LIN {X 0,Y 334.381,Z 572.13,A -85,B 0,C 180,E1 -16692.837,E2 -16692.837} C_VEL
LIN {X 0,Y 335.361,Z 549.408,A -85,B 0,C 180,E1 -16693.333,E2 -16693.333} C_VEL
LIN {X 0,Y 327.108,Z 531.714,A -85,B 0,C 180,E1 -16695.238,E2 -16695.238} C_VEL
LIN {X 0,Y 318.416,Z 515.187,A -85,B 0,C 180,E1 -16697.361,E2 -16697.361} C_VEL
LIN {X 0,Y 310.407,Z 501.402,A -85,B 0,C 180,E1 -16699.456,E2 -16699.456} C_VEL
LIN {X 0,Y 303.46,Z 490.565,A -85,B 0,C 180,E1 -16701.401,E2 -16701.401} C_VEL
LIN {X 0,Y 299.452,Z 484.565,A -85,B 0,C 180,E1 -16702.595,E2 -16702.595} C_VEL
LIN {X 0,Y 295.371,Z 478.736,A -85,B 0,C 180,E1 -16703.869,E2 -16703.869} C_VEL
LIN {X 0,Y 292.684,Z 474.795,A -85,B 0,C 180,E1 -16704.773,E2 -16704.773} C_VEL
LIN {X 0,Y 291.881,Z 473.268,A -85,B 0,C 180,E1 -16705.284,E2 -16705.284} C_VEL
LIN {X 0,Y 291.349,Z 471.542,A -85,B 0,C 180,E1 -16706.167,E2 -16706.167} C_VEL
LIN {X 0,Y 291.334,Z 471.401,A -85,B 0,C 180,E1 -16709.563,E2 -16709.563} C_VEL
LIN {X 0,Y 291.431,Z 471.376,A -85,B 0,C 180,E1 -16713.158,E2 -16713.158} C_VEL
LIN {X 0,Y 291.426,Z 471.42,A -85,B 0,C 180,E1 -16716.403,E2 -16716.403} C_VEL
LIN {X 0,Y 291.453,Z 471.349,A -85,B 0,C 180,E1 -16720.27,E2 -16720.27} C_VEL
LIN {X 0,Y 291.535,Z 471.417,A -85,B 0,C 180,E1 -16724.634,E2 -16724.634} C_VEL
LIN {X 0,Y 291.529,Z 471.42,A -85,B 0,C 180,E1 -16728.88,E2 -16728.88} C_VEL
LIN {X 0,Y 291.682,Z 471.379,A -85,B 0,C 180,E1 -16731.687,E2 -16731.687} C_VEL
LIN {X 0,Y 291.622,Z 471.406,A -85,B 0,C 180,E1 -16734.468,E2 -16734.468} C_VEL
LIN {X 0,Y 291.883,Z 471.376,A -85,B 0,C 180,E1 -16738.62,E2 -16738.62} C_VEL
LIN {X 0,Y 291.883,Z 471.351,A -85,B 0,C 180,E1 -16741.379,E2 -16741.379} C_VEL
LIN {X 0,Y 291.735,Z 471.371,A -85,B 0,C 180,E1 -16746.918,E2 -16746.918} C_VEL
LIN {X 0,Y 291.623,Z 471.396,A -85,B 0,C 180,E1 -16749.712,E2 -16749.712} C_VEL
LIN {X 0,Y 291.515,Z 471.42,A -85,B 0,C 180,E1 -16753.95,E2 -16753.95} C_VEL
LIN {X 0,Y 291.479,Z 471.41,A -85,B 0,C 180,E1 -16756.818,E2 -16756.818} C_VEL
LIN {X 0,Y 291.445,Z 471.415,A -85,B 0,C 180,E1 -16759.875,E2 -16759.875} C_VEL
LIN {X 0,Y 291.375,Z 471.402,A -85,B 0,C 180,E1 -16764.207,E2 -16764.207} C_VEL
LIN {X 0,Y 291.41,Z 471.367,A -85,B 0,C 180,E1 -16767.272,E2 -16767.272} C_VEL
LIN {X 0,Y 291.331,Z 471.448,A -85,B 0,C 180,E1 -16770.437,E2 -16770.437} C_VEL
LIN {X 0,Y 291.361,Z 471.384,A -85,B 0,C 180,E1 -16774.308,E2 -16774.308} C_VEL
LIN {X 0,Y 291.431,Z 471.801,A -85,B 0,C 180,E1 -16774.993,E2 -16774.993} C_VEL
LIN {X 0,Y 291.85,Z 473.233,A -85,B 0,C 180,E1 -16775.358,E2 -16775.358} C_VEL
LIN {X 0,Y 293.498,Z 475.642,A -85,B 0,C 180,E1 -16775.92,E2 -16775.92} C_VEL
LIN {X 0,Y 295.287,Z 477.12,A -85,B 0,C 180,E1 -16776.46,E2 -16776.46} C_VEL
LIN {X 0,Y 297.213,Z 480.287,A -85,B 0,C 180,E1 -16777.088,E2 -16777.088} C_VEL
LIN {X 0,Y 299.738,Z 482.814,A -85,B 0,C 180,E1 -16777.829,E2 -16777.829} C_VEL
LIN {X 0,Y 302.494,Z 486.373,A -85,B 0,C 180,E1 -16778.672,E2 -16778.672} C_VEL
LIN {X 0,Y 304.519,Z 488.28,A -85,B 0,C 180,E1 -16779.288,E2 -16779.288} C_VEL
LIN {X 0,Y 307.616,Z 492.007,A -85,B 0,C 180,E1 -16780.283,E2 -16780.283} C_VEL
LIN {X 0,Y 309.885,Z 494.075,A -85,B 0,C 180,E1 -16781.012,E2 -16781.012} C_VEL
LIN {X 0,Y 313.007,Z 497.745,A -85,B 0,C 180,E1 -16782.091,E2 -16782.091} C_VEL
LIN {X 0,Y 316.165,Z 500.564,A -85,B 0,C 180,E1 -16783.182,E2 -16783.182} C_VEL
LIN {X 0,Y 319.669,Z 504.411,A -85,B 0,C 180,E1 -16784.495,E2 -16784.495} C_VEL
LIN {X 0,Y 321.978,Z 506.47,A -85,B 0,C 180,E1 -16785.384,E2 -16785.384} C_VEL
LIN {X 0,Y 325.336,Z 510.246,A -85,B 0,C 180,E1 -16786.766,E2 -16786.766} C_VEL
LIN {X 0,Y 327.744,Z 512.477,A -85,B 0,C 180,E1 -16787.764,E2 -16787.764} C_VEL
LIN {X 0,Y 331.281,Z 516.359,A -85,B 0,C 180,E1 -16789.27,E2 -16789.27} C_VEL
LIN {X 0,Y 333.728,Z 518.535,A -85,B 0,C 180,E1 -16790.304,E2 -16790.304} C_VEL
LIN {X 0,Y 337.04,Z 522.208,A -85,B 0,C 180,E1 -16791.773,E2 -16791.773} C_VEL
LIN {X 0,Y 339.999,Z 524.765,A -85,B 0,C 180,E1 -16793.076,E2 -16793.076} C_VEL
LIN {X 0,Y 343.638,Z 528.709,A -85,B 0,C 180,E1 -16794.782,E2 -16794.782} C_VEL
LIN {X 0,Y 346.549,Z 531.16,A -85,B 0,C 180,E1 -16796.145,E2 -16796.145} C_VEL
LIN {X 0,Y 350.058,Z 534.897,A -85,B 0,C 180,E1 -16797.894,E2 -16797.894} C_VEL
LIN {X 0,Y 353.412,Z 537.55,A -85,B 0,C 180,E1 -16799.575,E2 -16799.575} C_VEL
LIN {X 0,Y 356.669,Z 541.059,A -85,B 0,C 180,E1 -16801.336,E2 -16801.336} C_VEL
LIN {X 0,Y 360.36,Z 544.044,A -85,B 0,C 180,E1 -16803.41,E2 -16803.41} C_VEL
LIN {X 0,Y 363.49,Z 547.556,A -85,B 0,C 180,E1 -16805.33,E2 -16805.33} C_VEL
LIN {X 0,Y 366.856,Z 549.992,A -85,B 0,C 180,E1 -16807.472,E2 -16807.472} C_VEL
LIN {X 0,Y 367.902,Z 550.793,A -85,B 0,C 180,E1 -16808.161,E2 -16808.161} C_VEL
LIN {X 0,Y 370.532,Z 553.885,A -85,B 0,C 180,E1 -16810.125,E2 -16810.125} C_VEL
LIN {X 0,Y 373.757,Z 556.298,A -85,B 0,C 180,E1 -16812.65,E2 -16812.65} C_VEL
LIN {X 0,Y 375.673,Z 557.433,A -85,B 0,C 180,E1 -16814.324,E2 -16814.324} C_VEL
LIN {X 0,Y 377.714,Z 560.107,A -85,B 0,C 180,E1 -16816.455,E2 -16816.455} C_VEL
LIN {X 0,Y 379.831,Z 562.032,A -85,B 0,C 180,E1 -16819.013,E2 -16819.013} C_VEL
LIN {X 0,Y 381.592,Z 562.974,A -85,B 0,C 180,E1 -16821.527,E2 -16821.527} C_VEL
LIN {X 0,Y 383.034,Z 563.727,A -85,B 0,C 180,E1 -16824.382,E2 -16824.382} C_VEL
LIN {X 0,Y 383.818,Z 564.175,A -85,B 0,C 180,E1 -16826.851,E2 -16826.851} C_VEL
LIN {X 0,Y 384.122,Z 564.361,A -85,B 0,C 180,E1 -16828.952,E2 -16828.952} C_VEL
LIN {X 0,Y 384.122,Z 564.364,A -85,B 0,C 180,E1 -16831.048,E2 -16831.048} C_VEL
LIN {X 0,Y 383.818,Z 564.175,A -85,B 0,C 180,E1 -16833.149,E2 -16833.149} C_VEL
LIN {X 0,Y 383.04,Z 563.678,A -85,B 0,C 180,E1 -16835.617,E2 -16835.617} C_VEL
LIN {X 0,Y 381.59,Z 562.994,A -85,B 0,C 180,E1 -16838.473,E2 -16838.473} C_VEL
LIN {X 0,Y 379.842,Z 561.96,A -85,B 0,C 180,E1 -16840.986,E2 -16840.986} C_VEL
LIN {X 0,Y 377.843,Z 560.265,A -85,B 0,C 180,E1 -16843.385,E2 -16843.385} C_VEL
LIN {X 0,Y 375.673,Z 557.437,A -85,B 0,C 180,E1 -16845.675,E2 -16845.675} C_VEL
LIN {X 0,Y 372.39,Z 555.413,A -85,B 0,C 180,E1 -16848.438,E2 -16848.438} C_VEL
LIN {X 0,Y 369.449,Z 552.788,A -85,B 0,C 180,E1 -16850.683,E2 -16850.683} C_VEL
LIN {X 0,Y 367.271,Z 550.225,A -85,B 0,C 180,E1 -16852.258,E2 -16852.258} C_VEL
LIN {X 0,Y 363.795,Z 547.809,A -85,B 0,C 180,E1 -16854.492,E2 -16854.492} C_VEL
LIN {X 0,Y 360.494,Z 544.264,A -85,B 0,C 180,E1 -16856.507,E2 -16856.507} C_VEL
LIN {X 0,Y 359.349,Z 543.135,A -85,B 0,C 180,E1 -16857.187,E2 -16857.187} C_VEL
LIN {X 0,Y 355.514,Z 540.032,A -85,B 0,C 180,E1 -16859.274,E2 -16859.274} C_VEL
LIN {X 0,Y 352.562,Z 536.779,A -85,B 0,C 180,E1 -16860.861,E2 -16860.861} C_VEL
LIN {X 0,Y 348.845,Z 533.753,A -85,B 0,C 180,E1 -16862.72,E2 -16862.72} C_VEL
LIN {X 0,Y 345.524,Z 530.115,A -85,B 0,C 180,E1 -16864.36,E2 -16864.36} C_VEL
LIN {X 0,Y 341.728,Z 526.843,A -85,B 0,C 180,E1 -16866.11,E2 -16866.11} C_VEL
LIN {X 0,Y 339.088,Z 523.809,A -85,B 0,C 180,E1 -16867.343,E2 -16867.343} C_VEL
LIN {X 0,Y 335.34,Z 520.521,A -85,B 0,C 180,E1 -16868.977,E2 -16868.977} C_VEL
LIN {X 0,Y 332.728,Z 517.523,A -85,B 0,C 180,E1 -16870.137,E2 -16870.137} C_VEL
LIN {X 0,Y 328.735,Z 513.73,A -85,B 0,C 180,E1 -16871.818,E2 -16871.818} C_VEL
LIN {X 0,Y 326.576,Z 511.305,A -85,B 0,C 180,E1 -16872.724,E2 -16872.724} C_VEL
LIN {X 0,Y 322.795,Z 507.577,A -85,B 0,C 180,E1 -16874.272,E2 -16874.272} C_VEL
LIN {X 0,Y 320.948,Z 505.42,A -85,B 0,C 180,E1 -16875.019,E2 -16875.019} C_VEL
LIN {X 0,Y 317.286,Z 501.993,A -85,B 0,C 180,E1 -16876.396,E2 -16876.396} C_VEL
LIN {X 0,Y 315.159,Z 499.492,A -85,B 0,C 180,E1 -16877.182,E2 -16877.182} C_VEL
LIN {X 0,Y 311.478,Z 496.114,A -85,B 0,C 180,E1 -16878.445,E2 -16878.445} C_VEL
LIN {X 0,Y 308.974,Z 493.165,A -85,B 0,C 180,E1 -16879.289,E2 -16879.289} C_VEL
LIN {X 0,Y 305.531,Z 489.71,A -85,B 0,C 180,E1 -16880.387,E2 -16880.387} C_VEL
LIN {X 0,Y 303.826,Z 487.508,A -85,B 0,C 180,E1 -16880.926,E2 -16880.926} C_VEL
LIN {X 0,Y 300.975,Z 484.659,A -85,B 0,C 180,E1 -16881.781,E2 -16881.781} C_VEL
LIN {X 0,Y 299.017,Z 481.929,A -85,B 0,C 180,E1 -16882.39,E2 -16882.39} C_VEL
LIN {X 0,Y 296.451,Z 479.267,A -85,B 0,C 180,E1 -16883.149,E2 -16883.149} C_VEL
LIN {X 0,Y 294.937,Z 476.731,A -85,B 0,C 180,E1 -16883.649,E2 -16883.649} C_VEL
LIN {X 0,Y 292.585,Z 474.553,A -85,B 0,C 180,E1 -16884.374,E2 -16884.374} C_VEL
LIN {X 0,Y 291.469,Z 471.949,A -85,B 0,C 180,E1 -16884.936,E2 -16884.936} C_VEL
LIN {X 0,Y 291.379,Z 471.439,A -85,B 0,C 180,E1 -16885.386,E2 -16885.386} C_VEL
LIN {X 0,Y 291.365,Z 471.403,A -85,B 0,C 180,E1 -16887.951,E2 -16887.951} C_VEL
LIN {X 0,Y 291.371,Z 471.396,A -85,B 0,C 180,E1 -16891.158,E2 -16891.158} C_VEL
LIN {X 0,Y 291.404,Z 471.37,A -85,B 0,C 180,E1 -16894.271,E2 -16894.271} C_VEL
LIN {X 0,Y 291.368,Z 471.442,A -85,B 0,C 180,E1 -16897.299,E2 -16897.299} C_VEL
LIN {X 0,Y 291.452,Z 471.414,A -85,B 0,C 180,E1 -16900.27,E2 -16900.27} C_VEL
LIN {X 0,Y 291.534,Z 471.399,A -85,B 0,C 180,E1 -16904.635,E2 -16904.635} C_VEL
LIN {X 0,Y 291.529,Z 471.397,A -85,B 0,C 180,E1 -16908.881,E2 -16908.881} C_VEL
LIN {X 0,Y 291.7,Z 471.394,A -85,B 0,C 180,E1 -16911.689,E2 -16911.689} C_VEL
LIN {X 0,Y 291.623,Z 471.389,A -85,B 0,C 180,E1 -16914.469,E2 -16914.469} C_VEL
LIN {X 0,Y 291.883,Z 471.353,A -85,B 0,C 180,E1 -16918.621,E2 -16918.621} C_VEL
LIN {X 0,Y 291.883,Z 471.377,A -85,B 0,C 180,E1 -16921.38,E2 -16921.38} C_VEL
LIN {X 0,Y 291.73,Z 471.386,A -85,B 0,C 180,E1 -16926.919,E2 -16926.919} C_VEL
LIN {X 0,Y 291.569,Z 471.399,A -85,B 0,C 180,E1 -16929.714,E2 -16929.714} C_VEL
LIN {X 0,Y 291.511,Z 471.402,A -85,B 0,C 180,E1 -16933.879,E2 -16933.879} C_VEL
LIN {X 0,Y 290.876,Z 471.497,A -85,B 0,C 180,E1 -16935.032,E2 -16935.032} C_VEL
LIN {X 0,Y 287.965,Z 471.838,A -85,B 0,C 180,E1 -16936.906,E2 -16936.906} C_VEL
LIN {X 0,Y 285.485,Z 472.113,A -85,B 0,C 180,E1 -16938.428,E2 -16938.428} C_VEL
LIN {X 0,Y 284.446,Z 472.222,A -85,B 0,C 180,E1 -16939.61,E2 -16939.61} C_VEL
LIN {X 0,Y 284.378,Z 472.229,A -85,B 0,C 180,E1 -16940.01,E2 -16940.01} C_VEL
LIN {X 0,Y 284.37,Z 472.306,A -85,B 0,C 180,E1 -16943.878,E2 -16943.878} C_VEL
LIN {X 0,Y 284.388,Z 472.248,A -85,B 0,C 180,E1 -16947.172,E2 -16947.172} C_VEL
LIN {X 0,Y 284.306,Z 472.298,A -85,B 0,C 180,E1 -16951.273,E2 -16951.273} C_VEL
LIN {X 0,Y 284.379,Z 472.631,A -85,B 0,C 180,E1 -16952.385,E2 -16952.385} C_VEL
LIN {X 0,Y 284.771,Z 474.121,A -85,B 0,C 180,E1 -16952.885,E2 -16952.885} C_VEL
LIN {X 0,Y 286.497,Z 476.648,A -85,B 0,C 180,E1 -16953.552,E2 -16953.552} C_VEL
LIN {X 0,Y 289.794,Z 480.785,A -85,B 0,C 180,E1 -16954.692,E2 -16954.692} C_VEL
LIN {X 0,Y 294.042,Z 486.894,A -85,B 0,C 180,E1 -16956.109,E2 -16956.109} C_VEL
LIN {X 0,Y 297.851,Z 492.54,A -85,B 0,C 180,E1 -16957.314,E2 -16957.314} C_VEL
LIN {X 0,Y 304.433,Z 502.659,A -85,B 0,C 180,E1 -16959.268,E2 -16959.268} C_VEL
LIN {X 0,Y 312.901,Z 517.15,A -85,B 0,C 180,E1 -16961.605,E2 -16961.605} C_VEL
LIN {X 0,Y 320.685,Z 531.778,A -85,B 0,C 180,E1 -16963.603,E2 -16963.603} C_VEL
LIN {X 0,Y 328.783,Z 548.886,A -85,B 0,C 180,E1 -16965.568,E2 -16965.568} C_VEL
LIN {X 0,Y 330.101,Z 551.932,A -85,B 0,C 180,E1 -16965.881,E2 -16965.881} C_VEL
LIN {X 0,Y 324.783,Z 665.436,A -85,B 0,C 180,E1 -16968.34,E2 -16968.34} C_VEL
LIN {X 0,Y 323.346,Z 691.603,A -85,B 0,C 180,E1 -16968.944,E2 -16968.944} C_VEL
LIN {X 0,Y 321.431,Z 710.108,A -85,B 0,C 180,E1 -16969.578,E2 -16969.578} C_VEL
LIN {X 0,Y 319.225,Z 725.277,A -85,B 0,C 180,E1 -16970.324,E2 -16970.324} C_VEL
LIN {X 0,Y 317.056,Z 738.026,A -85,B 0,C 180,E1 -16971.123,E2 -16971.123} C_VEL
LIN {X 0,Y 314.499,Z 750.717,A -85,B 0,C 180,E1 -16972.083,E2 -16972.083} C_VEL
LIN {X 0,Y 311.899,Z 762.357,A -85,B 0,C 180,E1 -16973.135,E2 -16973.135} C_VEL
LIN {X 0,Y 308.638,Z 775.182,A -85,B 0,C 180,E1 -16974.504,E2 -16974.504} C_VEL
LIN {X 0,Y 305.867,Z 785.571,A -85,B 0,C 180,E1 -16975.81,E2 -16975.81} C_VEL
LIN {X 0,Y 302.784,Z 796.148,A -85,B 0,C 180,E1 -16977.34,E2 -16977.34} C_VEL
LIN {X 0,Y 299.815,Z 805.837,A -85,B 0,C 180,E1 -16978.956,E2 -16978.956} C_VEL
LIN {X 0,Y 297.116,Z 814.636,A -85,B 0,C 180,E1 -16980.645,E2 -16980.645} C_VEL
LIN {X 0,Y 293.939,Z 825.009,A -85,B 0,C 180,E1 -16982.982,E2 -16982.982} C_VEL
LIN {X 0,Y 291.351,Z 832.898,A -85,B 0,C 180,E1 -16985.031,E2 -16985.031} C_VEL
LIN {X 0,Y 289.186,Z 839.864,A -85,B 0,C 180,E1 -16987.118,E2 -16987.118} C_VEL
LIN {X 0,Y 287.414,Z 846.008,A -85,B 0,C 180,E1 -16989.234,E2 -16989.234} C_VEL
LIN {X 0,Y 285.468,Z 852.957,A -85,B 0,C 180,E1 -16992.077,E2 -16992.077} C_VEL
LIN {X 0,Y 284.218,Z 858.207,A -85,B 0,C 180,E1 -16994.659,E2 -16994.659} C_VEL
LIN {X 0,Y 283.341,Z 862.335,A -85,B 0,C 180,E1 -16997.101,E2 -16997.101} C_VEL
LIN {X 0,Y 282.63,Z 866.188,A -85,B 0,C 180,E1 -16999.976,E2 -16999.976} C_VEL
LIN {X 0,Y 282.387,Z 869.045,A -85,B 0,C 180,E1 -17002.852,E2 -17002.852} C_VEL
LIN {X 0,Y 282.334,Z 870.439,A -85,B 0,C 180,E1 -17004.682,E2 -17004.682} C_VEL
LIN {X 0,Y 282.329,Z 871.61,A -85,B 0,C 180,E1 -17007.146,E2 -17007.146} C_VEL
LIN {X 0,Y 282.315,Z 872.083,A -85,B 0,C 180,E1 -17010,E2 -17010} C_VEL
LIN {X 0,Y 282.329,Z 871.61,A -85,B 0,C 180,E1 -17012.854,E2 -17012.854} C_VEL
LIN {X 0,Y 282.336,Z 870.182,A -85,B 0,C 180,E1 -17015.714,E2 -17015.714} C_VEL
LIN {X 0,Y 282.482,Z 867.793,A -85,B 0,C 180,E1 -17018.585,E2 -17018.585} C_VEL
LIN {X 0,Y 283.113,Z 863.375,A -85,B 0,C 180,E1 -17022.181,E2 -17022.181} C_VEL
LIN {X 0,Y 283.809,Z 860.006,A -85,B 0,C 180,E1 -17024.337,E2 -17024.337} C_VEL
LIN {X 0,Y 285.075,Z 854.503,A -85,B 0,C 180,E1 -17027.207,E2 -17027.207} C_VEL
LIN {X 0,Y 286.406,Z 849.643,A -85,B 0,C 180,E1 -17029.345,E2 -17029.345} C_VEL
LIN {X 0,Y 288.683,Z 841.563,A -85,B 0,C 180,E1 -17032.315,E2 -17032.315} C_VEL
LIN {X 0,Y 290.552,Z 835.315,A -85,B 0,C 180,E1 -17034.28,E2 -17034.28} C_VEL
LIN {X 0,Y 293.007,Z 827.765,A -85,B 0,C 180,E1 -17036.342,E2 -17036.342} C_VEL
LIN {X 0,Y 295.883,Z 818.635,A -85,B 0,C 180,E1 -17038.497,E2 -17038.497} C_VEL
LIN {X 0,Y 298.73,Z 809.388,A -85,B 0,C 180,E1 -17040.385,E2 -17040.385} C_VEL
LIN {X 0,Y 301.849,Z 799.167,A -85,B 0,C 180,E1 -17042.181,E2 -17042.181} C_VEL
LIN {X 0,Y 304.936,Z 788.746,A -85,B 0,C 180,E1 -17043.755,E2 -17043.755} C_VEL
LIN {X 0,Y 307.943,Z 777.792,A -85,B 0,C 180,E1 -17045.187,E2 -17045.187} C_VEL
LIN {X 0,Y 310.748,Z 766.854,A -85,B 0,C 180,E1 -17046.418,E2 -17046.418} C_VEL
LIN {X 0,Y 313.345,Z 755.941,A -85,B 0,C 180,E1 -17047.472,E2 -17047.472} C_VEL
LIN {X 0,Y 316.032,Z 743.211,A -85,B 0,C 180,E1 -17048.51,E2 -17048.51} C_VEL
LIN {X 0,Y 318.448,Z 730.004,A -85,B 0,C 180,E1 -17049.399,E2 -17049.399} C_VEL
LIN {X 0,Y 320.485,Z 717.004,A -85,B 0,C 180,E1 -17050.103,E2 -17050.103} C_VEL
LIN {X 0,Y 322.187,Z 703.636,A -85,B 0,C 180,E1 -17050.667,E2 -17050.667} C_VEL
LIN {X 0,Y 323.432,Z 690.183,A -85,B 0,C 180,E1 -17051.094,E2 -17051.094} C_VEL
LIN {X 0,Y 325.351,Z 652.898,A -85,B 0,C 180,E1 -17051.934,E2 -17051.934} C_VEL
LIN {X 0,Y 330.17,Z 552.059,A -85,B 0,C 180,E1 -17054.104,E2 -17054.104} C_VEL
LIN {X 0,Y 322.6,Z 535.681,A -85,B 0,C 180,E1 -17055.922,E2 -17055.922} C_VEL
LIN {X 0,Y 314.412,Z 519.91,A -85,B 0,C 180,E1 -17057.996,E2 -17057.996} C_VEL
LIN {X 0,Y 306.931,Z 506.798,A -85,B 0,C 180,E1 -17060.022,E2 -17060.022} C_VEL
LIN {X 0,Y 300.04,Z 495.907,A -85,B 0,C 180,E1 -17062.018,E2 -17062.018} C_VEL
LIN {X 0,Y 296.102,Z 489.901,A -85,B 0,C 180,E1 -17063.234,E2 -17063.234} C_VEL
LIN {X 0,Y 292.28,Z 484.386,A -85,B 0,C 180,E1 -17064.467,E2 -17064.467} C_VEL
LIN {X 0,Y 288.574,Z 479.142,A -85,B 0,C 180,E1 -17065.728,E2 -17065.728} C_VEL
LIN {X 0,Y 284.924,Z 474.496,A -85,B 0,C 180,E1 -17067.041,E2 -17067.041} C_VEL
LIN {X 0,Y 284.431,Z 472.918,A -85,B 0,C 180,E1 -17067.477,E2 -17067.477} C_VEL
LIN {X 0,Y 284.376,Z 472.392,A -85,B 0,C 180,E1 -17067.903,E2 -17067.903} C_VEL
LIN {X 0,Y 284.321,Z 472.249,A -85,B 0,C 180,E1 -17071.988,E2 -17071.988} C_VEL
LIN {X 0,Y 284.347,Z 472.31,A -85,B 0,C 180,E1 -17075.154,E2 -17075.154} C_VEL
LIN {X 0,Y 284.31,Z 472.252,A -85,B 0,C 180,E1 -17078.235,E2 -17078.235} C_VEL
LIN {X 0,Y 284.392,Z 472.236,A -85,B 0,C 180,E1 -17081.261,E2 -17081.261} C_VEL
LIN {X 0,Y 284.473,Z 472.298,A -85,B 0,C 180,E1 -17084.469,E2 -17084.469} C_VEL
LIN {X 0,Y 284.481,Z 472.294,A -85,B 0,C 180,E1 -17088.601,E2 -17088.601} C_VEL
LIN {X 0,Y 284.633,Z 472.256,A -85,B 0,C 180,E1 -17091.48,E2 -17091.48} C_VEL
LIN {X 0,Y 284.593,Z 472.283,A -85,B 0,C 180,E1 -17094.331,E2 -17094.331} C_VEL
LIN {X 0,Y 284.849,Z 472.251,A -85,B 0,C 180,E1 -17098.586,E2 -17098.586} C_VEL
LIN {X 0,Y 284.849,Z 472.226,A -85,B 0,C 180,E1 -17101.413,E2 -17101.413} C_VEL
LIN {X 0,Y 284.688,Z 472.249,A -85,B 0,C 180,E1 -17107.09,E2 -17107.09} C_VEL
LIN {X 0,Y 284.56,Z 472.271,A -85,B 0,C 180,E1 -17109.955,E2 -17109.955} C_VEL
LIN {X 0,Y 284.472,Z 472.29,A -85,B 0,C 180,E1 -17114.303,E2 -17114.303} C_VEL
LIN {X 0,Y 284.416,Z 472.295,A -85,B 0,C 180,E1 -17117.248,E2 -17117.248} C_VEL
LIN {X 0,Y 284.371,Z 472.294,A -85,B 0,C 180,E1 -17120.242,E2 -17120.242} C_VEL
LIN {X 0,Y 284.329,Z 472.262,A -85,B 0,C 180,E1 -17124.847,E2 -17124.847} C_VEL
LIN {X 0,Y 284.319,Z 472.256,A -85,B 0,C 180,E1 -17128.011,E2 -17128.011} C_VEL
LIN {X 0,Y 284.345,Z 472.276,A -85,B 0,C 180,E1 -17132.041,E2 -17132.041} C_VEL
LIN {X 0,Y 284.336,Z 472.559,A -85,B 0,C 180,E1 -17132.821,E2 -17132.821} C_VEL
LIN {X 0,Y 284.661,Z 473.798,A -85,B 0,C 180,E1 -17133.268,E2 -17133.268} C_VEL
LIN {X 0,Y 286.187,Z 476.255,A -85,B 0,C 180,E1 -17133.858,E2 -17133.858} C_VEL
LIN {X 0,Y 288.455,Z 478.173,A -85,B 0,C 180,E1 -17134.612,E2 -17134.612} C_VEL
LIN {X 0,Y 290.288,Z 481.161,A -85,B 0,C 180,E1 -17135.263,E2 -17135.263} C_VEL
LIN {X 0,Y 292.472,Z 483.386,A -85,B 0,C 180,E1 -17135.96,E2 -17135.96} C_VEL
LIN {X 0,Y 295.096,Z 487.032,A -85,B 0,C 180,E1 -17136.808,E2 -17136.808} C_VEL
LIN {X 0,Y 296.858,Z 488.838,A -85,B 0,C 180,E1 -17137.334,E2 -17137.334} C_VEL
LIN {X 0,Y 299.815,Z 492.532,A -85,B 0,C 180,E1 -17138.232,E2 -17138.232} C_VEL
LIN {X 0,Y 301.873,Z 494.497,A -85,B 0,C 180,E1 -17138.836,E2 -17138.836} C_VEL
LIN {X 0,Y 305.432,Z 498.533,A -85,B 0,C 180,E1 -17139.95,E2 -17139.95} C_VEL
LIN {X 0,Y 307.628,Z 500.638,A -85,B 0,C 180,E1 -17140.646,E2 -17140.646} C_VEL
LIN {X 0,Y 311.443,Z 504.735,A -85,B 0,C 180,E1 -17141.927,E2 -17141.927} C_VEL
LIN {X 0,Y 314.013,Z 507.046,A -85,B 0,C 180,E1 -17142.798,E2 -17142.798} C_VEL
LIN {X 0,Y 317.607,Z 510.88,A -85,B 0,C 180,E1 -17144.118,E2 -17144.118} C_VEL
LIN {X 0,Y 319.983,Z 512.995,A -85,B 0,C 180,E1 -17145.011,E2 -17145.011} C_VEL
LIN {X 0,Y 323.545,Z 516.875,A -85,B 0,C 180,E1 -17146.453,E2 -17146.453} C_VEL
LIN {X 0,Y 325.996,Z 519.227,A -85,B 0,C 180,E1 -17147.459,E2 -17147.459} C_VEL
LIN {X 0,Y 329.92,Z 523.309,A -85,B 0,C 180,E1 -17149.112,E2 -17149.112} C_VEL
LIN {X 0,Y 331.953,Z 525.148,A -85,B 0,C 180,E1 -17149.958,E2 -17149.958} C_VEL
LIN {X 0,Y 335.766,Z 529.203,A -85,B 0,C 180,E1 -17151.636,E2 -17151.636} C_VEL
LIN {X 0,Y 338.425,Z 531.541,A -85,B 0,C 180,E1 -17152.804,E2 -17152.804} C_VEL
LIN {X 0,Y 342.225,Z 535.55,A -85,B 0,C 180,E1 -17154.564,E2 -17154.564} C_VEL
LIN {X 0,Y 345.179,Z 538.054,A -85,B 0,C 180,E1 -17155.94,E2 -17155.94} C_VEL
LIN {X 0,Y 348.729,Z 541.782,A -85,B 0,C 180,E1 -17157.702,E2 -17157.702} C_VEL
LIN {X 0,Y 351.946,Z 544.324,A -85,B 0,C 180,E1 -17159.307,E2 -17159.307} C_VEL
LIN {X 0,Y 355.165,Z 547.781,A -85,B 0,C 180,E1 -17161.037,E2 -17161.037} C_VEL
LIN {X 0,Y 359.171,Z 551.025,A -85,B 0,C 180,E1 -17163.254,E2 -17163.254} C_VEL
LIN {X 0,Y 362.444,Z 554.622,A -85,B 0,C 180,E1 -17165.254,E2 -17165.254} C_VEL
LIN {X 0,Y 366.069,Z 557.131,A -85,B 0,C 180,E1 -17167.544,E2 -17167.544} C_VEL
LIN {X 0,Y 369.45,Z 560.835,A -85,B 0,C 180,E1 -17169.977,E2 -17169.977} C_VEL
LIN {X 0,Y 372.6,Z 563.185,A -85,B 0,C 180,E1 -17172.435,E2 -17172.435} C_VEL
LIN {X 0,Y 374.66,Z 564.449,A -85,B 0,C 180,E1 -17174.201,E2 -17174.201} C_VEL
LIN {X 0,Y 376.8,Z 567.179,A -85,B 0,C 180,E1 -17176.421,E2 -17176.421} C_VEL
LIN {X 0,Y 378.934,Z 569.079,A -85,B 0,C 180,E1 -17178.987,E2 -17178.987} C_VEL
LIN {X 0,Y 380.71,Z 570.019,A -85,B 0,C 180,E1 -17181.508,E2 -17181.508} C_VEL
LIN {X 0,Y 382.002,Z 570.622,A -85,B 0,C 180,E1 -17184.011,E2 -17184.011} C_VEL
LIN {X 0,Y 382.654,Z 571.132,A -85,B 0,C 180,E1 -17185.787,E2 -17185.787} C_VEL
LIN {X 0,Y 383.151,Z 571.293,A -85,B 0,C 180,E1 -17187.898,E2 -17187.898} C_VEL
LIN {X 0,Y 383.34,Z 571.349,A -85,B 0,C 180,E1 -17190,E2 -17190} C_VEL
LIN {X 0,Y 383.151,Z 571.294,A -85,B 0,C 180,E1 -17192.102,E2 -17192.102} C_VEL
LIN {X 0,Y 382.496,Z 571.028,A -85,B 0,C 180,E1 -17194.694,E2 -17194.694} C_VEL
LIN {X 0,Y 381.321,Z 570.322,A -85,B 0,C 180,E1 -17197.412,E2 -17197.412} C_VEL
LIN {X 0,Y 379.645,Z 569.506,A -85,B 0,C 180,E1 -17200.07,E2 -17200.07} C_VEL
LIN {X 0,Y 377.507,Z 567.926,A -85,B 0,C 180,E1 -17202.74,E2 -17202.74} C_VEL
LIN {X 0,Y 375.425,Z 565.498,A -85,B 0,C 180,E1 -17205.035,E2 -17205.035} C_VEL
LIN {X 0,Y 374.396,Z 564.104,A -85,B 0,C 180,E1 -17206.05,E2 -17206.05} C_VEL
LIN {X 0,Y 371.444,Z 562.454,A -85,B 0,C 180,E1 -17208.487,E2 -17208.487} C_VEL
LIN {X 0,Y 368.378,Z 559.8,A -85,B 0,C 180,E1 -17210.8,E2 -17210.8} C_VEL
LIN {X 0,Y 366.07,Z 557.136,A -85,B 0,C 180,E1 -17212.457,E2 -17212.457} C_VEL
LIN {X 0,Y 362.446,Z 554.612,A -85,B 0,C 180,E1 -17214.747,E2 -17214.747} C_VEL
LIN {X 0,Y 359.063,Z 550.952,A -85,B 0,C 180,E1 -17216.81,E2 -17216.81} C_VEL
LIN {X 0,Y 357.753,Z 549.797,A -85,B 0,C 180,E1 -17217.555,E2 -17217.555} C_VEL
LIN {X 0,Y 353.873,Z 546.58,A -85,B 0,C 180,E1 -17219.658,E2 -17219.658} C_VEL
LIN {X 0,Y 351.189,Z 543.603,A -85,B 0,C 180,E1 -17221.088,E2 -17221.088} C_VEL
LIN {X 0,Y 347.28,Z 540.406,A -85,B 0,C 180,E1 -17223.021,E2 -17223.021} C_VEL
LIN {X 0,Y 343.964,Z 536.89,A -85,B 0,C 180,E1 -17224.633,E2 -17224.633} C_VEL
LIN {X 0,Y 339.964,Z 533.38,A -85,B 0,C 180,E1 -17226.47,E2 -17226.47} C_VEL
LIN {X 0,Y 337.366,Z 530.449,A -85,B 0,C 180,E1 -17227.664,E2 -17227.664} C_VEL
LIN {X 0,Y 333.548,Z 527.09,A -85,B 0,C 180,E1 -17229.322,E2 -17229.322} C_VEL
LIN {X 0,Y 331.011,Z 524.2,A -85,B 0,C 180,E1 -17230.438,E2 -17230.438} C_VEL
LIN {X 0,Y 327.099,Z 520.525,A -85,B 0,C 180,E1 -17232.073,E2 -17232.073} C_VEL
LIN {X 0,Y 324.66,Z 517.809,A -85,B 0,C 180,E1 -17233.105,E2 -17233.105} C_VEL
LIN {X 0,Y 320.712,Z 513.934,A -85,B 0,C 180,E1 -17234.695,E2 -17234.695} C_VEL
LIN {X 0,Y 318.781,Z 511.796,A -85,B 0,C 180,E1 -17235.455,E2 -17235.455} C_VEL
LIN {X 0,Y 314.829,Z 508.059,A -85,B 0,C 180,E1 -17236.899,E2 -17236.899} C_VEL
LIN {X 0,Y 312.794,Z 505.825,A -85,B 0,C 180,E1 -17237.62,E2 -17237.62} C_VEL
LIN {X 0,Y 308.869,Z 502.157,A -85,B 0,C 180,E1 -17238.936,E2 -17238.936} C_VEL
LIN {X 0,Y 306.435,Z 499.394,A -85,B 0,C 180,E1 -17239.737,E2 -17239.737} C_VEL
LIN {X 0,Y 302.72,Z 495.657,A -85,B 0,C 180,E1 -17240.891,E2 -17240.891} C_VEL
LIN {X 0,Y 300.986,Z 493.546,A -85,B 0,C 180,E1 -17241.432,E2 -17241.432} C_VEL
LIN {X 0,Y 297.587,Z 489.944,A -85,B 0,C 180,E1 -17242.438,E2 -17242.438} C_VEL
LIN {X 0,Y 295.872,Z 487.752,A -85,B 0,C 180,E1 -17242.962,E2 -17242.962} C_VEL
LIN {X 0,Y 293.13,Z 484.531,A -85,B 0,C 180,E1 -17243.815,E2 -17243.815} C_VEL
LIN {X 0,Y 292.021,Z 482.764,A -85,B 0,C 180,E1 -17244.189,E2 -17244.189} C_VEL
LIN {X 0,Y 289.471,Z 480.074,A -85,B 0,C 180,E1 -17245.015,E2 -17245.015} C_VEL
LIN {X 0,Y 288.027,Z 477.677,A -85,B 0,C 180,E1 -17245.534,E2 -17245.534} C_VEL
LIN {X 0,Y 285.644,Z 475.624,A -85,B 0,C 180,E1 -17246.334,E2 -17246.334} C_VEL
LIN {X 0,Y 284.393,Z 472.94,A -85,B 0,C 180,E1 -17246.961,E2 -17246.961} C_VEL
LIN {X 0,Y 284.31,Z 472.32,A -85,B 0,C 180,E1 -17247.446,E2 -17247.446} C_VEL
LIN {X 0,Y 284.352,Z 472.29,A -85,B 0,C 180,E1 -17250.376,E2 -17250.376} C_VEL
LIN {X 0,Y 284.367,Z 472.24,A -85,B 0,C 180,E1 -17253.586,E2 -17253.586} C_VEL
LIN {X 0,Y 284.327,Z 472.306,A -85,B 0,C 180,E1 -17256.704,E2 -17256.704} C_VEL
LIN {X 0,Y 284.393,Z 472.305,A -85,B 0,C 180,E1 -17261.261,E2 -17261.261} C_VEL
LIN {X 0,Y 284.472,Z 472.278,A -85,B 0,C 180,E1 -17264.47,E2 -17264.47} C_VEL
LIN {X 0,Y 284.481,Z 472.274,A -85,B 0,C 180,E1 -17268.602,E2 -17268.602} C_VEL
LIN {X 0,Y 284.65,Z 472.274,A -85,B 0,C 180,E1 -17271.481,E2 -17271.481} C_VEL
LIN {X 0,Y 284.593,Z 472.263,A -85,B 0,C 180,E1 -17274.331,E2 -17274.331} C_VEL
LIN {X 0,Y 284.849,Z 472.229,A -85,B 0,C 180,E1 -17278.587,E2 -17278.587} C_VEL
LIN {X 0,Y 284.849,Z 472.253,A -85,B 0,C 180,E1 -17281.414,E2 -17281.414} C_VEL
LIN {X 0,Y 284.681,Z 472.261,A -85,B 0,C 180,E1 -17287.091,E2 -17287.091} C_VEL
LIN {X 0,Y 284.513,Z 472.28,A -85,B 0,C 180,E1 -17289.957,E2 -17289.957} C_VEL
LIN {X 0,Y 284.472,Z 472.282,A -85,B 0,C 180,E1 -17294.303,E2 -17294.303} C_VEL
LIN {X 0,Y 284.417,Z 472.267,A -85,B 0,C 180,E1 -17297.249,E2 -17297.249} C_VEL
LIN {X 0,Y 284.378,Z 472.229,A -85,B 0,C 180,E1 -17300.01,E2 -17300.01} C_VEL
LIN {X 0,Y 283.743,Z 472.319,A -85,B 0,C 180,E1 -17301.193,E2 -17301.193} C_VEL
LIN {X 0,Y 280.867,Z 472.714,A -85,B 0,C 180,E1 -17303.119,E2 -17303.119} C_VEL
LIN {X 0,Y 278.414,Z 473.052,A -85,B 0,C 180,E1 -17304.683,E2 -17304.683} C_VEL
LIN {X 0,Y 277.376,Z 473.146,A -85,B 0,C 180,E1 -17305.896,E2 -17305.896} C_VEL
LIN {X 0,Y 277.302,Z 473.143,A -85,B 0,C 180,E1 -17306.307,E2 -17306.307} C_VEL
LIN {X 0,Y 277.308,Z 473.311,A -85,B 0,C 180,E1 -17310.036,E2 -17310.036} C_VEL
LIN {X 0,Y 277.499,Z 474.28,A -85,B 0,C 180,E1 -17310.495,E2 -17310.495} C_VEL
LIN {X 0,Y 279.005,Z 477.022,A -85,B 0,C 180,E1 -17311.195,E2 -17311.195} C_VEL
LIN {X 0,Y 281.492,Z 479.087,A -85,B 0,C 180,E1 -17312.111,E2 -17312.111} C_VEL
LIN {X 0,Y 283.387,Z 482.182,A -85,B 0,C 180,E1 -17312.853,E2 -17312.853} C_VEL
LIN {X 0,Y 286.842,Z 486.535,A -85,B 0,C 180,E1 -17314.088,E2 -17314.088} C_VEL
LIN {X 0,Y 291.131,Z 492.765,A -85,B 0,C 180,E1 -17315.565,E2 -17315.565} C_VEL
LIN {X 0,Y 294.993,Z 498.661,A -85,B 0,C 180,E1 -17316.828,E2 -17316.828} C_VEL
LIN {X 0,Y 301.438,Z 508.787,A -85,B 0,C 180,E1 -17318.799,E2 -17318.799} C_VEL
LIN {X 0,Y 309.143,Z 522.237,A -85,B 0,C 180,E1 -17320.997,E2 -17320.997} C_VEL
LIN {X 0,Y 316.753,Z 536.757,A -85,B 0,C 180,E1 -17323.018,E2 -17323.018} C_VEL
LIN {X 0,Y 324.404,Z 553.16,A -85,B 0,C 180,E1 -17324.941,E2 -17324.941} C_VEL
LIN {X 0,Y 324.895,Z 554.301,A -85,B 0,C 180,E1 -17325.062,E2 -17325.062} C_VEL
LIN {X 0,Y 319.63,Z 663.437,A -85,B 0,C 180,E1 -17327.459,E2 -17327.459} C_VEL
LIN {X 0,Y 318.024,Z 691.393,A -85,B 0,C 180,E1 -17328.103,E2 -17328.103} C_VEL
LIN {X 0,Y 316.048,Z 709.898,A -85,B 0,C 180,E1 -17328.742,E2 -17328.742} C_VEL
LIN {X 0,Y 313.781,Z 725.067,A -85,B 0,C 180,E1 -17329.494,E2 -17329.494} C_VEL
LIN {X 0,Y 311.442,Z 738.342,A -85,B 0,C 180,E1 -17330.339,E2 -17330.339} C_VEL
LIN {X 0,Y 308.898,Z 750.506,A -85,B 0,C 180,E1 -17331.269,E2 -17331.269} C_VEL
LIN {X 0,Y 306.184,Z 762.145,A -85,B 0,C 180,E1 -17332.329,E2 -17332.329} C_VEL
LIN {X 0,Y 302.85,Z 774.971,A -85,B 0,C 180,E1 -17333.719,E2 -17333.719} C_VEL
LIN {X 0,Y 299.674,Z 786.281,A -85,B 0,C 180,E1 -17335.167,E2 -17335.167} C_VEL
LIN {X 0,Y 296.44,Z 796.942,A -85,B 0,C 180,E1 -17336.754,E2 -17336.754} C_VEL
LIN {X 0,Y 293.081,Z 807.399,A -85,B 0,C 180,E1 -17338.564,E2 -17338.564} C_VEL
LIN {X 0,Y 290.373,Z 815.833,A -85,B 0,C 180,E1 -17340.254,E2 -17340.254} C_VEL
LIN {X 0,Y 287.511,Z 824.795,A -85,B 0,C 180,E1 -17342.327,E2 -17342.327} C_VEL
LIN {X 0,Y 284.798,Z 832.684,A -85,B 0,C 180,E1 -17344.416,E2 -17344.416} C_VEL
LIN {X 0,Y 282.544,Z 839.65,A -85,B 0,C 180,E1 -17346.548,E2 -17346.548} C_VEL
LIN {X 0,Y 280.673,Z 845.794,A -85,B 0,C 180,E1 -17348.711,E2 -17348.711} C_VEL
LIN {X 0,Y 278.624,Z 852.744,A -85,B 0,C 180,E1 -17351.622,E2 -17351.622} C_VEL
LIN {X 0,Y 277.191,Z 858.342,A -85,B 0,C 180,E1 -17354.465,E2 -17354.465} C_VEL
LIN {X 0,Y 276.322,Z 862.122,A -85,B 0,C 180,E1 -17356.768,E2 -17356.768} C_VEL
LIN {X 0,Y 275.572,Z 865.976,A -85,B 0,C 180,E1 -17359.716,E2 -17359.716} C_VEL
LIN {X 0,Y 275.294,Z 868.833,A -85,B 0,C 180,E1 -17362.667,E2 -17362.667} C_VEL
LIN {X 0,Y 275.238,Z 870.332,A -85,B 0,C 180,E1 -17364.768,E2 -17364.768} C_VEL
LIN {X 0,Y 275.239,Z 871.4,A -85,B 0,C 180,E1 -17367.073,E2 -17367.073} C_VEL
LIN {X 0,Y 275.238,Z 871.874,A -85,B 0,C 180,E1 -17370,E2 -17370} C_VEL
LIN {X 0,Y 275.239,Z 871.4,A -85,B 0,C 180,E1 -17372.927,E2 -17372.927} C_VEL
LIN {X 0,Y 275.235,Z 869.971,A -85,B 0,C 180,E1 -17375.862,E2 -17375.862} C_VEL
LIN {X 0,Y 275.402,Z 867.581,A -85,B 0,C 180,E1 -17378.807,E2 -17378.807} C_VEL
LIN {X 0,Y 276.09,Z 863.163,A -85,B 0,C 180,E1 -17382.496,E2 -17382.496} C_VEL
LIN {X 0,Y 276.836,Z 859.794,A -85,B 0,C 180,E1 -17384.706,E2 -17384.706} C_VEL
LIN {X 0,Y 278.181,Z 854.289,A -85,B 0,C 180,E1 -17387.648,E2 -17387.648} C_VEL
LIN {X 0,Y 279.615,Z 849.43,A -85,B 0,C 180,E1 -17389.835,E2 -17389.835} C_VEL
LIN {X 0,Y 282.075,Z 841.135,A -85,B 0,C 180,E1 -17392.946,E2 -17392.946} C_VEL
LIN {X 0,Y 284.403,Z 833.893,A -85,B 0,C 180,E1 -17395.231,E2 -17395.231} C_VEL
LIN {X 0,Y 286.588,Z 827.553,A -85,B 0,C 180,E1 -17396.979,E2 -17396.979} C_VEL
LIN {X 0,Y 289.387,Z 818.966,A -85,B 0,C 180,E1 -17399.059,E2 -17399.059} C_VEL
LIN {X 0,Y 292.529,Z 809.175,A -85,B 0,C 180,E1 -17401.099,E2 -17401.099} C_VEL
LIN {X 0,Y 295.799,Z 798.955,A -85,B 0,C 180,E1 -17402.921,E2 -17402.921} C_VEL
LIN {X 0,Y 299.05,Z 788.344,A -85,B 0,C 180,E1 -17404.546,E2 -17404.546} C_VEL
LIN {X 0,Y 302.113,Z 777.58,A -85,B 0,C 180,E1 -17405.971,E2 -17405.971} C_VEL
LIN {X 0,Y 305.016,Z 766.643,A -85,B 0,C 180,E1 -17407.216,E2 -17407.216} C_VEL
LIN {X 0,Y 308.089,Z 753.988,A -85,B 0,C 180,E1 -17408.433,E2 -17408.433} C_VEL
LIN {X 0,Y 310.723,Z 741.818,A -85,B 0,C 180,E1 -17409.414,E2 -17409.414} C_VEL
LIN {X 0,Y 313.01,Z 729.634,A -85,B 0,C 180,E1 -17410.235,E2 -17410.235} C_VEL
LIN {X 0,Y 315.092,Z 716.795,A -85,B 0,C 180,E1 -17410.933,E2 -17410.933} C_VEL
LIN {X 0,Y 316.833,Z 703.426,A -85,B 0,C 180,E1 -17411.504,E2 -17411.504} C_VEL
LIN {X 0,Y 318.117,Z 689.973,A -85,B 0,C 180,E1 -17411.935,E2 -17411.935} C_VEL
LIN {X 0,Y 320.113,Z 652.688,A -85,B 0,C 180,E1 -17412.782,E2 -17412.782} C_VEL
LIN {X 0,Y 324.928,Z 555.451,A -85,B 0,C 180,E1 -17414.897,E2 -17414.897} C_VEL
LIN {X 0,Y 324.729,Z 553.936,A -85,B 0,C 180,E1 -17414.978,E2 -17414.978} C_VEL
LIN {X 0,Y 317.416,Z 538.122,A -85,B 0,C 180,E1 -17416.81,E2 -17416.81} C_VEL
LIN {X 0,Y 309.143,Z 522.174,A -85,B 0,C 180,E1 -17419.005,E2 -17419.005} C_VEL
LIN {X 0,Y 302.519,Z 510.706,A -85,B 0,C 180,E1 -17420.878,E2 -17420.878} C_VEL
LIN {X 0,Y 296.656,Z 501.24,A -85,B 0,C 180,E1 -17422.648,E2 -17422.648} C_VEL
LIN {X 0,Y 293.046,Z 495.627,A -85,B 0,C 180,E1 -17423.802,E2 -17423.802} C_VEL
LIN {X 0,Y 289.2,Z 489.973,A -85,B 0,C 180,E1 -17425.087,E2 -17425.087} C_VEL
LIN {X 0,Y 285.657,Z 484.879,A -85,B 0,C 180,E1 -17426.335,E2 -17426.335} C_VEL
LIN {X 0,Y 281.981,Z 480.094,A -85,B 0,C 180,E1 -17427.686,E2 -17427.686} C_VEL
LIN {X 0,Y 281.042,Z 478.652,A -85,B 0,C 180,E1 -17428.055,E2 -17428.055} C_VEL
LIN {X 0,Y 278.591,Z 476.503,A -85,B 0,C 180,E1 -17428.97,E2 -17428.97} C_VEL
LIN {X 0,Y 277.371,Z 473.785,A -85,B 0,C 180,E1 -17429.67,E2 -17429.67} C_VEL
LIN {X 0,Y 277.314,Z 473.212,A -85,B 0,C 180,E1 -17430.175,E2 -17430.175} C_VEL
LIN {X 0,Y 277.35,Z 473.123,A -85,B 0,C 180,E1 -17432.863,E2 -17432.863} C_VEL
LIN {X 0,Y 277.33,Z 473.181,A -85,B 0,C 180,E1 -17436.079,E2 -17436.079} C_VEL
LIN {X 0,Y 277.336,Z 473.107,A -85,B 0,C 180,E1 -17440.765,E2 -17440.765} C_VEL
LIN {X 0,Y 277.422,Z 473.163,A -85,B 0,C 180,E1 -17445.325,E2 -17445.325} C_VEL
LIN {X 0,Y 277.455,Z 473.164,A -85,B 0,C 180,E1 -17449.787,E2 -17449.787} C_VEL
LIN {X 0,Y 277.635,Z 473.136,A -85,B 0,C 180,E1 -17452.728,E2 -17452.728} C_VEL
LIN {X 0,Y 277.815,Z 473.127,A -85,B 0,C 180,E1 -17458.55,E2 -17458.55} C_VEL
LIN {X 0,Y 277.815,Z 473.102,A -85,B 0,C 180,E1 -17461.449,E2 -17461.449} C_VEL
LIN {X 0,Y 277.643,Z 473.127,A -85,B 0,C 180,E1 -17467.271,E2 -17467.271} C_VEL
LIN {X 0,Y 277.5,Z 473.147,A -85,B 0,C 180,E1 -17470.211,E2 -17470.211} C_VEL
LIN {X 0,Y 277.422,Z 473.162,A -85,B 0,C 180,E1 -17474.674,E2 -17474.674} C_VEL
LIN {X 0,Y 277.336,Z 473.177,A -85,B 0,C 180,E1 -17479.234,E2 -17479.234} C_VEL
LIN {X 0,Y 277.284,Z 473.153,A -85,B 0,C 180,E1 -17484.157,E2 -17484.157} C_VEL
LIN {X 0,Y 277.315,Z 473.121,A -85,B 0,C 180,E1 -17487.503,E2 -17487.503} C_VEL
LIN {X 0,Y 277.287,Z 473.389,A -85,B 0,C 180,E1 -17490.489,E2 -17490.489} C_VEL
LIN {X 0,Y 277.601,Z 474.66,A -85,B 0,C 180,E1 -17490.999,E2 -17490.999} C_VEL
LIN {X 0,Y 279.02,Z 477.019,A -85,B 0,C 180,E1 -17491.615,E2 -17491.615} C_VEL
LIN {X 0,Y 281.542,Z 479.122,A -85,B 0,C 180,E1 -17492.545,E2 -17492.545} C_VEL
LIN {X 0,Y 283.626,Z 482.38,A -85,B 0,C 180,E1 -17493.352,E2 -17493.352} C_VEL
LIN {X 0,Y 285.725,Z 484.389,A -85,B 0,C 180,E1 -17494.08,E2 -17494.08} C_VEL
LIN {X 0,Y 288.222,Z 487.901,A -85,B 0,C 180,E1 -17494.963,E2 -17494.963} C_VEL
LIN {X 0,Y 289.685,Z 489.502,A -85,B 0,C 180,E1 -17495.445,E2 -17495.445} C_VEL
LIN {X 0,Y 292.582,Z 493.333,A -85,B 0,C 180,E1 -17496.397,E2 -17496.397} C_VEL
LIN {X 0,Y 294.387,Z 495.454,A -85,B 0,C 180,E1 -17496.959,E2 -17496.959} C_VEL
LIN {X 0,Y 298.024,Z 499.48,A -85,B 0,C 180,E1 -17498.047,E2 -17498.047} C_VEL
LIN {X 0,Y 303.048,Z 504.908,A -85,B 0,C 180,E1 -17499.57,E2 -17499.57} C_VEL
LIN {X 0,Y 305.218,Z 507.007,A -85,B 0,C 180,E1 -17500.242,E2 -17500.242} C_VEL
LIN {X 0,Y 309.393,Z 511.312,A -85,B 0,C 180,E1 -17501.6,E2 -17501.6} C_VEL
LIN {X 0,Y 311.746,Z 513.456,A -85,B 0,C 180,E1 -17502.401,E2 -17502.401} C_VEL
LIN {X 0,Y 315.836,Z 517.601,A -85,B 0,C 180,E1 -17503.855,E2 -17503.855} C_VEL
LIN {X 0,Y 318.251,Z 519.817,A -85,B 0,C 180,E1 -17504.746,E2 -17504.746} C_VEL
LIN {X 0,Y 321.932,Z 523.686,A -85,B 0,C 180,E1 -17506.21,E2 -17506.21} C_VEL
LIN {X 0,Y 324.172,Z 525.828,A -85,B 0,C 180,E1 -17507.115,E2 -17507.115} C_VEL
LIN {X 0,Y 328.3,Z 530.045,A -85,B 0,C 180,E1 -17508.843,E2 -17508.843} C_VEL
LIN {X 0,Y 330.207,Z 531.826,A -85,B 0,C 180,E1 -17509.647,E2 -17509.647} C_VEL
LIN {X 0,Y 334.282,Z 536.029,A -85,B 0,C 180,E1 -17511.411,E2 -17511.411} C_VEL
LIN {X 0,Y 336.708,Z 538.152,A -85,B 0,C 180,E1 -17512.481,E2 -17512.481} C_VEL
LIN {X 0,Y 340.613,Z 542.233,A -85,B 0,C 180,E1 -17514.265,E2 -17514.265} C_VEL
LIN {X 0,Y 343.71,Z 544.906,A -85,B 0,C 180,E1 -17515.699,E2 -17515.699} C_VEL
LIN {X 0,Y 347.661,Z 548.887,A -85,B 0,C 180,E1 -17517.639,E2 -17517.639} C_VEL
LIN {X 0,Y 350.568,Z 551.185,A -85,B 0,C 180,E1 -17519.081,E2 -17519.081} C_VEL
LIN {X 0,Y 353.948,Z 554.715,A -85,B 0,C 180,E1 -17520.886,E2 -17520.886} C_VEL
LIN {X 0,Y 357.77,Z 557.762,A -85,B 0,C 180,E1 -17522.973,E2 -17522.973} C_VEL
LIN {X 0,Y 361.22,Z 561.502,A -85,B 0,C 180,E1 -17525.068,E2 -17525.068} C_VEL
LIN {X 0,Y 364.673,Z 563.914,A -85,B 0,C 180,E1 -17527.211,E2 -17527.211} C_VEL
LIN {X 0,Y 366.386,Z 565.677,A -85,B 0,C 180,E1 -17528.38,E2 -17528.38} C_VEL
LIN {X 0,Y 369.126,Z 568.443,A -85,B 0,C 180,E1 -17530.42,E2 -17530.42} C_VEL
LIN {X 0,Y 372.071,Z 570.452,A -85,B 0,C 180,E1 -17532.717,E2 -17532.717} C_VEL
LIN {X 0,Y 373.636,Z 571.441,A -85,B 0,C 180,E1 -17534.076,E2 -17534.076} C_VEL
LIN {X 0,Y 375.81,Z 574.176,A -85,B 0,C 180,E1 -17536.315,E2 -17536.315} C_VEL
LIN {X 0,Y 377.972,Z 576.078,A -85,B 0,C 180,E1 -17538.879,E2 -17538.879} C_VEL
LIN {X 0,Y 379.828,Z 577.064,A -85,B 0,C 180,E1 -17541.488,E2 -17541.488} C_VEL
LIN {X 0,Y 381.128,Z 577.671,A -85,B 0,C 180,E1 -17543.997,E2 -17543.997} C_VEL
LIN {X 0,Y 381.783,Z 578.177,A -85,B 0,C 180,E1 -17545.777,E2 -17545.777} C_VEL
LIN {X 0,Y 382.286,Z 578.339,A -85,B 0,C 180,E1 -17547.893,E2 -17547.893} C_VEL
LIN {X 0,Y 382.474,Z 578.396,A -85,B 0,C 180,E1 -17550,E2 -17550} C_VEL
LIN {X 0,Y 382.286,Z 578.341,A -85,B 0,C 180,E1 -17552.107,E2 -17552.107} C_VEL
LIN {X 0,Y 381.626,Z 578.074,A -85,B 0,C 180,E1 -17554.705,E2 -17554.705} C_VEL
LIN {X 0,Y 380.445,Z 577.364,A -85,B 0,C 180,E1 -17557.43,E2 -17557.43} C_VEL
LIN {X 0,Y 378.757,Z 576.552,A -85,B 0,C 180,E1 -17560.094,E2 -17560.094} C_VEL
LIN {X 0,Y 376.601,Z 574.98,A -85,B 0,C 180,E1 -17562.771,E2 -17562.771} C_VEL
LIN {X 0,Y 374.407,Z 572.489,A -85,B 0,C 180,E1 -17565.156,E2 -17565.156} C_VEL
LIN {X 0,Y 373.103,Z 570.953,A -85,B 0,C 180,E1 -17566.412,E2 -17566.412} C_VEL
LIN {X 0,Y 370.127,Z 569.192,A -85,B 0,C 180,E1 -17568.832,E2 -17568.832} C_VEL
LIN {X 0,Y 367.121,Z 566.584,A -85,B 0,C 180,E1 -17571.059,E2 -17571.059} C_VEL
LIN {X 0,Y 364.871,Z 564.035,A -85,B 0,C 180,E1 -17572.658,E2 -17572.658} C_VEL
LIN {X 0,Y 361.224,Z 561.489,A -85,B 0,C 180,E1 -17574.933,E2 -17574.933} C_VEL
LIN {X 0,Y 357.875,Z 557.945,A -85,B 0,C 180,E1 -17576.961,E2 -17576.961} C_VEL
LIN {X 0,Y 356.403,Z 556.608,A -85,B 0,C 180,E1 -17577.789,E2 -17577.789} C_VEL
LIN {X 0,Y 352.644,Z 553.522,A -85,B 0,C 180,E1 -17579.817,E2 -17579.817} C_VEL
LIN {X 0,Y 349.773,Z 550.394,A -85,B 0,C 180,E1 -17581.338,E2 -17581.338} C_VEL
LIN {X 0,Y 345.769,Z 547.153,A -85,B 0,C 180,E1 -17583.283,E2 -17583.283} C_VEL
LIN {X 0,Y 342.383,Z 543.609,A -85,B 0,C 180,E1 -17584.92,E2 -17584.92} C_VEL
LIN {X 0,Y 338.187,Z 539.887,A -85,B 0,C 180,E1 -17586.846,E2 -17586.846} C_VEL
LIN {X 0,Y 335.523,Z 537.017,A -85,B 0,C 180,E1 -17588.045,E2 -17588.045} C_VEL
LIN {X 0,Y 331.508,Z 533.325,A -85,B 0,C 180,E1 -17589.79,E2 -17589.79} C_VEL
LIN {X 0,Y 328.907,Z 530.529,A -85,B 0,C 180,E1 -17590.902,E2 -17590.902} C_VEL
LIN {X 0,Y 324.909,Z 526.7,A -85,B 0,C 180,E1 -17592.568,E2 -17592.568} C_VEL
LIN {X 0,Y 322.594,Z 524.23,A -85,B 0,C 180,E1 -17593.527,E2 -17593.527} C_VEL
LIN {X 0,Y 318.747,Z 520.454,A -85,B 0,C 180,E1 -17595.056,E2 -17595.056} C_VEL
LIN {X 0,Y 316.908,Z 518.445,A -85,B 0,C 180,E1 -17595.761,E2 -17595.761} C_VEL
LIN {X 0,Y 312.637,Z 514.472,A -85,B 0,C 180,E1 -17597.292,E2 -17597.292} C_VEL
LIN {X 0,Y 310.302,Z 512.055,A -85,B 0,C 180,E1 -17598.095,E2 -17598.095} C_VEL
LIN {X 0,Y 306.128,Z 508.063,A -85,B 0,C 180,E1 -17599.465,E2 -17599.465} C_VEL
LIN {X 0,Y 303.879,Z 505.608,A -85,B 0,C 180,E1 -17600.183,E2 -17600.183} C_VEL
LIN {X 0,Y 299.77,Z 501.456,A -85,B 0,C 180,E1 -17601.431,E2 -17601.431} C_VEL
LIN {X 0,Y 297.848,Z 499.339,A -85,B 0,C 180,E1 -17602.004,E2 -17602.004} C_VEL
LIN {X 0,Y 294.183,Z 495.163,A -85,B 0,C 180,E1 -17603.106,E2 -17603.106} C_VEL
LIN {X 0,Y 289.934,Z 489.933,A -85,B 0,C 180,E1 -17604.467,E2 -17604.467} C_VEL
LIN {X 0,Y 288.819,Z 488.48,A -85,B 0,C 180,E1 -17604.842,E2 -17604.842} C_VEL
LIN {X 0,Y 286.139,Z 485.146,A -85,B 0,C 180,E1 -17605.764,E2 -17605.764} C_VEL
LIN {X 0,Y 285.178,Z 483.763,A -85,B 0,C 180,E1 -17606.112,E2 -17606.112} C_VEL
LIN {X 0,Y 282.635,Z 481.119,A -85,B 0,C 180,E1 -17607.015,E2 -17607.015} C_VEL
LIN {X 0,Y 281.154,Z 478.646,A -85,B 0,C 180,E1 -17607.603,E2 -17607.603} C_VEL
LIN {X 0,Y 278.613,Z 476.538,A -85,B 0,C 180,E1 -17608.545,E2 -17608.545} C_VEL
LIN {X 0,Y 277.439,Z 474.193,A -85,B 0,C 180,E1 -17609.14,E2 -17609.14} C_VEL
LIN {X 0,Y 277.261,Z 473.275,A -85,B 0,C 180,E1 -17609.659,E2 -17609.659} C_VEL
LIN {X 0,Y 277.348,Z 473.114,A -85,B 0,C 180,E1 -17612.864,E2 -17612.864} C_VEL
LIN {X 0,Y 277.29,Z 473.159,A -85,B 0,C 180,E1 -17616.076,E2 -17616.076} C_VEL
LIN {X 0,Y 277.336,Z 473.176,A -85,B 0,C 180,E1 -17620.766,E2 -17620.766} C_VEL
LIN {X 0,Y 277.422,Z 473.162,A -85,B 0,C 180,E1 -17625.326,E2 -17625.326} C_VEL
LIN {X 0,Y 277.5,Z 473.148,A -85,B 0,C 180,E1 -17629.789,E2 -17629.789} C_VEL
LIN {X 0,Y 277.643,Z 473.13,A -85,B 0,C 180,E1 -17632.729,E2 -17632.729} C_VEL
LIN {X 0,Y 277.815,Z 473.105,A -85,B 0,C 180,E1 -17638.551,E2 -17638.551} C_VEL
LIN {X 0,Y 277.815,Z 473.128,A -85,B 0,C 180,E1 -17641.45,E2 -17641.45} C_VEL
LIN {X 0,Y 277.635,Z 473.135,A -85,B 0,C 180,E1 -17647.272,E2 -17647.272} C_VEL
LIN {X 0,Y 277.455,Z 473.163,A -85,B 0,C 180,E1 -17650.213,E2 -17650.213} C_VEL
LIN {X 0,Y 277.422,Z 473.164,A -85,B 0,C 180,E1 -17654.675,E2 -17654.675} C_VEL
LIN {X 0,Y 277.336,Z 473.108,A -85,B 0,C 180,E1 -17659.235,E2 -17659.235} C_VEL
LIN {X 0,Y 277.32,Z 473.191,A -85,B 0,C 180,E1 -17664.173,E2 -17664.173} C_VEL
LIN {X 0,Y 277.302,Z 473.143,A -85,B 0,C 180,E1 -17666.307,E2 -17666.307} C_VEL
LIN {X 0,Y 277.266,Z 473.516,A -85,B 0,C 180,E1 -17667.11,E2 -17667.11} C_VEL
LIN {X 0,Y 277.139,Z 475.255,A -85,B 0,C 180,E1 -17668.272,E2 -17668.272} C_VEL
LIN {X 0,Y 277.158,Z 477.962,A -85,B 0,C 180,E1 -17669.362,E2 -17669.362} C_VEL
LIN {X 0,Y 277.857,Z 482.472,A -85,B 0,C 180,E1 -17670.732,E2 -17670.732} C_VEL
LIN {X 0,Y 279.267,Z 486.011,A -85,B 0,C 180,E1 -17671.691,E2 -17671.691} C_VEL
LIN {X 0,Y 279.971,Z 487.148,A -85,B 0,C 180,E1 -17671.998,E2 -17671.998} C_VEL
LIN {X 0,Y 284.057,Z 492.461,A -85,B 0,C 180,E1 -17673.521,E2 -17673.521} C_VEL
LIN {X 0,Y 288.23,Z 498.671,A -85,B 0,C 180,E1 -17675.008,E2 -17675.008} C_VEL
LIN {X 0,Y 291.918,Z 504.384,A -85,B 0,C 180,E1 -17676.253,E2 -17676.253} C_VEL
LIN {X 0,Y 297.92,Z 513.967,A -85,B 0,C 180,E1 -17678.153,E2 -17678.153} C_VEL
LIN {X 0,Y 305.333,Z 527.076,A -85,B 0,C 180,E1 -17680.345,E2 -17680.345} C_VEL
LIN {X 0,Y 312.88,Z 541.767,A -85,B 0,C 180,E1 -17682.425,E2 -17682.425} C_VEL
LIN {X 0,Y 319.837,Z 556.934,A -85,B 0,C 180,E1 -17684.24,E2 -17684.24} C_VEL
LIN {X 0,Y 313.504,Z 681.137,A -85,B 0,C 180,E1 -17686.975,E2 -17686.975} C_VEL
LIN {X 0,Y 312.125,Z 698.22,A -85,B 0,C 180,E1 -17687.454,E2 -17687.454} C_VEL
LIN {X 0,Y 310.26,Z 712.751,A -85,B 0,C 180,E1 -17688.016,E2 -17688.016} C_VEL
LIN {X 0,Y 308.39,Z 724.856,A -85,B 0,C 180,E1 -17688.633,E2 -17688.633} C_VEL
LIN {X 0,Y 306.201,Z 737.037,A -85,B 0,C 180,E1 -17689.406,E2 -17689.406} C_VEL
LIN {X 0,Y 303.358,Z 750.295,A -85,B 0,C 180,E1 -17690.425,E2 -17690.425} C_VEL
LIN {X 0,Y 300.543,Z 761.933,A -85,B 0,C 180,E1 -17691.494,E2 -17691.494} C_VEL
LIN {X 0,Y 297.11,Z 774.759,A -85,B 0,C 180,E1 -17692.902,E2 -17692.902} C_VEL
LIN {X 0,Y 293.861,Z 785.957,A -85,B 0,C 180,E1 -17694.354,E2 -17694.354} C_VEL
LIN {X 0,Y 290.502,Z 796.732,A -85,B 0,C 180,E1 -17695.983,E2 -17695.983} C_VEL
LIN {X 0,Y 286.974,Z 807.187,A -85,B 0,C 180,E1 -17697.816,E2 -17697.816} C_VEL
LIN {X 0,Y 284.14,Z 815.62,A -85,B 0,C 180,E1 -17699.533,E2 -17699.533} C_VEL
LIN {X 0,Y 281.113,Z 824.581,A -85,B 0,C 180,E1 -17701.641,E2 -17701.641} C_VEL
LIN {X 0,Y 278.301,Z 832.471,A -85,B 0,C 180,E1 -17703.773,E2 -17703.773} C_VEL
LIN {X 0,Y 275.923,Z 839.436,A -85,B 0,C 180,E1 -17705.951,E2 -17705.951} C_VEL
LIN {X 0,Y 273.945,Z 845.581,A -85,B 0,C 180,E1 -17708.162,E2 -17708.162} C_VEL
LIN {X 0,Y 271.78,Z 852.531,A -85,B 0,C 180,E1 -17711.142,E2 -17711.142} C_VEL
LIN {X 0,Y 270.55,Z 857.006,A -85,B 0,C 180,E1 -17713.397,E2 -17713.397} C_VEL
LIN {X 0,Y 269.322,Z 861.91,A -85,B 0,C 180,E1 -17716.417,E2 -17716.417} C_VEL
LIN {X 0,Y 268.511,Z 865.764,A -85,B 0,C 180,E1 -17719.443,E2 -17719.443} C_VEL
LIN {X 0,Y 268.225,Z 868.623,A -85,B 0,C 180,E1 -17722.472,E2 -17722.472} C_VEL
LIN {X 0,Y 268.13,Z 870.512,A -85,B 0,C 180,E1 -17725.49,E2 -17725.49} C_VEL
LIN {X 0,Y 268.151,Z 871.19,A -85,B 0,C 180,E1 -17726.995,E2 -17726.995} C_VEL
LIN {X 0,Y 268.164,Z 871.665,A -85,B 0,C 180,E1 -17730,E2 -17730} C_VEL
LIN {X 0,Y 268.15,Z 871.19,A -85,B 0,C 180,E1 -17733.005,E2 -17733.005} C_VEL
LIN {X 0,Y 268.144,Z 869.761,A -85,B 0,C 180,E1 -17736.018,E2 -17736.018} C_VEL
LIN {X 0,Y 268.34,Z 867.37,A -85,B 0,C 180,E1 -17739.041,E2 -17739.041} C_VEL
LIN {X 0,Y 269.076,Z 862.95,A -85,B 0,C 180,E1 -17742.827,E2 -17742.827} C_VEL
LIN {X 0,Y 269.883,Z 859.581,A -85,B 0,C 180,E1 -17745.094,E2 -17745.094} C_VEL
LIN {X 0,Y 271.335,Z 854.077,A -85,B 0,C 180,E1 -17748.108,E2 -17748.108} C_VEL
LIN {X 0,Y 272.814,Z 849.216,A -85,B 0,C 180,E1 -17750.351,E2 -17750.351} C_VEL
LIN {X 0,Y 275.273,Z 841.398,A -85,B 0,C 180,E1 -17753.366,E2 -17753.366} C_VEL
LIN {X 0,Y 277.469,Z 834.889,A -85,B 0,C 180,E1 -17755.505,E2 -17755.505} C_VEL
LIN {X 0,Y 280.199,Z 827.34,A -85,B 0,C 180,E1 -17757.646,E2 -17757.646} C_VEL
LIN {X 0,Y 283.1,Z 818.753,A -85,B 0,C 180,E1 -17759.768,E2 -17759.768} C_VEL
LIN {X 0,Y 286.392,Z 808.963,A -85,B 0,C 180,E1 -17761.843,E2 -17761.843} C_VEL
LIN {X 0,Y 289.791,Z 798.742,A -85,B 0,C 180,E1 -17763.693,E2 -17763.693} C_VEL
LIN {X 0,Y 293.166,Z 788.147,A -85,B 0,C 180,E1 -17765.339,E2 -17765.339} C_VEL
LIN {X 0,Y 296.334,Z 777.368,A -85,B 0,C 180,E1 -17766.786,E2 -17766.786} C_VEL
LIN {X 0,Y 299.351,Z 766.431,A -85,B 0,C 180,E1 -17768.044,E2 -17768.044} C_VEL
LIN {X 0,Y 302.512,Z 753.776,A -85,B 0,C 180,E1 -17769.276,E2 -17769.276} C_VEL
LIN {X 0,Y 305.228,Z 741.729,A -85,B 0,C 180,E1 -17770.255,E2 -17770.255} C_VEL
LIN {X 0,Y 307.626,Z 729.254,A -85,B 0,C 180,E1 -17771.104,E2 -17771.104} C_VEL
LIN {X 0,Y 309.754,Z 716.584,A -85,B 0,C 180,E1 -17771.795,E2 -17771.795} C_VEL
LIN {X 0,Y 311.54,Z 703.216,A -85,B 0,C 180,E1 -17772.371,E2 -17772.371} C_VEL
LIN {X 0,Y 312.879,Z 689.763,A -85,B 0,C 180,E1 -17772.802,E2 -17772.802} C_VEL
LIN {X 0,Y 314.94,Z 652.478,A -85,B 0,C 180,E1 -17773.659,E2 -17773.659} C_VEL
LIN {X 0,Y 319.838,Z 556.922,A -85,B 0,C 180,E1 -17775.76,E2 -17775.76} C_VEL
LIN {X 0,Y 312.116,Z 540.242,A -85,B 0,C 180,E1 -17777.779,E2 -17777.779} C_VEL
LIN {X 0,Y 304.034,Z 524.686,A -85,B 0,C 180,E1 -17780.027,E2 -17780.027} C_VEL
LIN {X 0,Y 296.777,Z 512.069,A -85,B 0,C 180,E1 -17782.199,E2 -17782.199} C_VEL
LIN {X 0,Y 289.828,Z 501.062,A -85,B 0,C 180,E1 -17784.448,E2 -17784.448} C_VEL
LIN {X 0,Y 286.281,Z 495.73,A -85,B 0,C 180,E1 -17785.676,E2 -17785.676} C_VEL
LIN {X 0,Y 282.386,Z 490.133,A -85,B 0,C 180,E1 -17787.096,E2 -17787.096} C_VEL
LIN {X 0,Y 279.227,Z 485.921,A -85,B 0,C 180,E1 -17788.304,E2 -17788.304} C_VEL
LIN {X 0,Y 278.414,Z 484.857,A -85,B 0,C 180,E1 -17788.625,E2 -17788.625} C_VEL
LIN {X 0,Y 275.824,Z 482.194,A -85,B 0,C 180,E1 -17789.645,E2 -17789.645} C_VEL
LIN {X 0,Y 274.381,Z 479.624,A -85,B 0,C 180,E1 -17790.291,E2 -17790.291} C_VEL
LIN {X 0,Y 271.869,Z 477.742,A -85,B 0,C 180,E1 -17791.325,E2 -17791.325} C_VEL
LIN {X 0,Y 270.438,Z 474.961,A -85,B 0,C 180,E1 -17792.11,E2 -17792.11} C_VEL
LIN {X 0,Y 270.3,Z 474.073,A -85,B 0,C 180,E1 -17792.725,E2 -17792.725} C_VEL
LIN {X 0,Y 270.224,Z 474.03,A -85,B 0,C 180,E1 -17797.038,E2 -17797.038} C_VEL
LIN {X 0,Y 270.294,Z 473.979,A -85,B 0,C 180,E1 -17800.244,E2 -17800.244} C_VEL
LIN {X 0,Y 270.391,Z 474.045,A -85,B 0,C 180,E1 -17804.934,E2 -17804.934} C_VEL
LIN {X 0,Y 270.407,Z 474.046,A -85,B 0,C 180,E1 -17809.517,E2 -17809.517} C_VEL
LIN {X 0,Y 270.593,Z 474.011,A -85,B 0,C 180,E1 -17812.538,E2 -17812.538} C_VEL
LIN {X 0,Y 270.781,Z 474.003,A -85,B 0,C 180,E1 -17818.512,E2 -17818.512} C_VEL
LIN {X 0,Y 270.781,Z 473.978,A -85,B 0,C 180,E1 -17821.487,E2 -17821.487} C_VEL
LIN {X 0,Y 270.602,Z 474.006,A -85,B 0,C 180,E1 -17827.461,E2 -17827.461} C_VEL
LIN {X 0,Y 270.435,Z 474.024,A -85,B 0,C 180,E1 -17830.481,E2 -17830.481} C_VEL
LIN {X 0,Y 270.39,Z 474.034,A -85,B 0,C 180,E1 -17835.065,E2 -17835.065} C_VEL
LIN {X 0,Y 270.294,Z 474.048,A -85,B 0,C 180,E1 -17839.756,E2 -17839.756} C_VEL
LIN {X 0,Y 270.231,Z 474.019,A -85,B 0,C 180,E1 -17844.589,E2 -17844.589} C_VEL
LIN {X 0,Y 270.264,Z 474.14,A -85,B 0,C 180,E1 -17847.807,E2 -17847.807} C_VEL
LIN {X 0,Y 270.528,Z 475.325,A -85,B 0,C 180,E1 -17848.407,E2 -17848.407} C_VEL
LIN {X 0,Y 271.975,Z 477.879,A -85,B 0,C 180,E1 -17849.139,E2 -17849.139} C_VEL
LIN {X 0,Y 274.707,Z 480.141,A -85,B 0,C 180,E1 -17850.269,E2 -17850.269} C_VEL
LIN {X 0,Y 276.661,Z 483.268,A -85,B 0,C 180,E1 -17851.117,E2 -17851.117} C_VEL
LIN {X 0,Y 279.089,Z 485.58,A -85,B 0,C 180,E1 -17852.05,E2 -17852.05} C_VEL
LIN {X 0,Y 281.452,Z 488.889,A -85,B 0,C 180,E1 -17852.97,E2 -17852.97} C_VEL
LIN {X 0,Y 283.138,Z 490.672,A -85,B 0,C 180,E1 -17853.577,E2 -17853.577} C_VEL
LIN {X 0,Y 286.129,Z 494.547,A -85,B 0,C 180,E1 -17854.644,E2 -17854.644} C_VEL
LIN {X 0,Y 290.087,Z 499.635,A -85,B 0,C 180,E1 -17855.98,E2 -17855.98} C_VEL
LIN {X 0,Y 295.147,Z 505.491,A -85,B 0,C 180,E1 -17857.552,E2 -17857.552} C_VEL
LIN {X 0,Y 300.7,Z 511.331,A -85,B 0,C 180,E1 -17859.207,E2 -17859.207} C_VEL
LIN {X 0,Y 303.562,Z 514.23,A -85,B 0,C 180,E1 -17860.083,E2 -17860.083} C_VEL
LIN {X 0,Y 308.086,Z 518.506,A -85,B 0,C 180,E1 -17861.533,E2 -17861.533} C_VEL
LIN {X 0,Y 313.757,Z 524.094,A -85,B 0,C 180,E1 -17863.488,E2 -17863.488} C_VEL
LIN {X 0,Y 316.289,Z 526.434,A -85,B 0,C 180,E1 -17864.405,E2 -17864.405} C_VEL
LIN {X 0,Y 320.339,Z 530.499,A -85,B 0,C 180,E1 -17865.977,E2 -17865.977} C_VEL
LIN {X 0,Y 322.228,Z 532.322,A -85,B 0,C 180,E1 -17866.735,E2 -17866.735} C_VEL
LIN {X 0,Y 326.642,Z 536.757,A -85,B 0,C 180,E1 -17868.56,E2 -17868.56} C_VEL
LIN {X 0,Y 328.625,Z 538.71,A -85,B 0,C 180,E1 -17869.407,E2 -17869.407} C_VEL
LIN {X 0,Y 332.861,Z 542.926,A -85,B 0,C 180,E1 -17871.226,E2 -17871.226} C_VEL
LIN {X 0,Y 335.196,Z 545.033,A -85,B 0,C 180,E1 -17872.25,E2 -17872.25} C_VEL
LIN {X 0,Y 339.126,Z 549.023,A -85,B 0,C 180,E1 -17874.03,E2 -17874.03} C_VEL
LIN {X 0,Y 342.067,Z 551.544,A -85,B 0,C 180,E1 -17875.385,E2 -17875.385} C_VEL
LIN {X 0,Y 346.181,Z 555.637,A -85,B 0,C 180,E1 -17877.368,E2 -17877.368} C_VEL
LIN {X 0,Y 349.275,Z 558.171,A -85,B 0,C 180,E1 -17878.903,E2 -17878.903} C_VEL
LIN {X 0,Y 352.786,Z 561.693,A -85,B 0,C 180,E1 -17880.762,E2 -17880.762} C_VEL
LIN {X 0,Y 356.576,Z 564.773,A -85,B 0,C 180,E1 -17882.817,E2 -17882.817} C_VEL
LIN {X 0,Y 359.944,Z 568.345,A -85,B 0,C 180,E1 -17884.847,E2 -17884.847} C_VEL
LIN {X 0,Y 363.475,Z 570.808,A -85,B 0,C 180,E1 -17887.009,E2 -17887.009} C_VEL
LIN {X 0,Y 365.164,Z 572.586,A -85,B 0,C 180,E1 -17888.179,E2 -17888.179} C_VEL
LIN {X 0,Y 368.162,Z 575.491,A -85,B 0,C 180,E1 -17890.366,E2 -17890.366} C_VEL
LIN {X 0,Y 371.125,Z 577.483,A -85,B 0,C 180,E1 -17892.671,E2 -17892.671} C_VEL
LIN {X 0,Y 372.607,Z 578.43,A -85,B 0,C 180,E1 -17893.951,E2 -17893.951} C_VEL
LIN {X 0,Y 374.623,Z 580.967,A -85,B 0,C 180,E1 -17896.003,E2 -17896.003} C_VEL
LIN {X 0,Y 376.902,Z 582.99,A -85,B 0,C 180,E1 -17898.631,E2 -17898.631} C_VEL
LIN {X 0,Y 378.752,Z 583.974,A -85,B 0,C 180,E1 -17901.153,E2 -17901.153} C_VEL
LIN {X 0,Y 380.102,Z 584.645,A -85,B 0,C 180,E1 -17903.631,E2 -17903.631} C_VEL
LIN {X 0,Y 380.912,Z 585.222,A -85,B 0,C 180,E1 -17905.768,E2 -17905.768} C_VEL
LIN {X 0,Y 381.421,Z 585.385,A -85,B 0,C 180,E1 -17907.888,E2 -17907.888} C_VEL
LIN {X 0,Y 381.609,Z 585.442,A -85,B 0,C 180,E1 -17910,E2 -17910} C_VEL
LIN {X 0,Y 381.421,Z 585.387,A -85,B 0,C 180,E1 -17912.112,E2 -17912.112} C_VEL
LIN {X 0,Y 380.774,Z 585.101,A -85,B 0,C 180,E1 -17914.673,E2 -17914.673} C_VEL
LIN {X 0,Y 379.568,Z 584.408,A -85,B 0,C 180,E1 -17917.447,E2 -17917.447} C_VEL
LIN {X 0,Y 377.778,Z 583.516,A -85,B 0,C 180,E1 -17920.252,E2 -17920.252} C_VEL
LIN {X 0,Y 375.696,Z 582.031,A -85,B 0,C 180,E1 -17922.802,E2 -17922.802} C_VEL
LIN {X 0,Y 373.474,Z 579.599,A -85,B 0,C 180,E1 -17925.195,E2 -17925.195} C_VEL
LIN {X 0,Y 372.175,Z 577.966,A -85,B 0,C 180,E1 -17926.454,E2 -17926.454} C_VEL
LIN {X 0,Y 369.162,Z 576.244,A -85,B 0,C 180,E1 -17928.883,E2 -17928.883} C_VEL
LIN {X 0,Y 366.037,Z 573.566,A -85,B 0,C 180,E1 -17931.192,E2 -17931.192} C_VEL
LIN {X 0,Y 363.678,Z 570.945,A -85,B 0,C 180,E1 -17932.857,E2 -17932.857} C_VEL
LIN {X 0,Y 359.948,Z 568.334,A -85,B 0,C 180,E1 -17935.154,E2 -17935.154} C_VEL
LIN {X 0,Y 356.339,Z 564.509,A -85,B 0,C 180,E1 -17937.318,E2 -17937.318} C_VEL
LIN {X 0,Y 351.62,Z 560.67,A -85,B 0,C 180,E1 -17939.865,E2 -17939.865} C_VEL
LIN {X 0,Y 348.17,Z 557.111,A -85,B 0,C 180,E1 -17941.656,E2 -17941.656} C_VEL
LIN {X 0,Y 344.18,Z 553.804,A -85,B 0,C 180,E1 -17943.591,E2 -17943.591} C_VEL
LIN {X 0,Y 340.483,Z 550.073,A -85,B 0,C 180,E1 -17945.363,E2 -17945.363} C_VEL
LIN {X 0,Y 336.038,Z 546.037,A -85,B 0,C 180,E1 -17947.37,E2 -17947.37} C_VEL
LIN {X 0,Y 333.833,Z 543.664,A -85,B 0,C 180,E1 -17948.363,E2 -17948.363} C_VEL
LIN {X 0,Y 329.765,Z 539.967,A -85,B 0,C 180,E1 -17950.111,E2 -17950.111} C_VEL
LIN {X 0,Y 326.877,Z 536.947,A -85,B 0,C 180,E1 -17951.343,E2 -17951.343} C_VEL
LIN {X 0,Y 322.594,Z 532.76,A -85,B 0,C 180,E1 -17953.112,E2 -17953.112} C_VEL
LIN {X 0,Y 320.34,Z 530.485,A -85,B 0,C 180,E1 -17954.023,E2 -17954.023} C_VEL
LIN {X 0,Y 316.183,Z 526.342,A -85,B 0,C 180,E1 -17955.633,E2 -17955.633} C_VEL
LIN {X 0,Y 313.986,Z 524.272,A -85,B 0,C 180,E1 -17956.43,E2 -17956.43} C_VEL
LIN {X 0,Y 309.72,Z 520.098,A -85,B 0,C 180,E1 -17957.915,E2 -17957.915} C_VEL
LIN {X 0,Y 303.784,Z 514.497,A -85,B 0,C 180,E1 -17959.844,E2 -17959.844} C_VEL
LIN {X 0,Y 300.876,Z 511.471,A -85,B 0,C 180,E1 -17960.741,E2 -17960.741} C_VEL
LIN {X 0,Y 296.593,Z 507.022,A -85,B 0,C 180,E1 -17962.023,E2 -17962.023} C_VEL
LIN {X 0,Y 291.496,Z 501.369,A -85,B 0,C 180,E1 -17963.567,E2 -17963.567} C_VEL
LIN {X 0,Y 286.847,Z 495.451,A -85,B 0,C 180,E1 -17965.108,E2 -17965.108} C_VEL
LIN {X 0,Y 283.137,Z 490.684,A -85,B 0,C 180,E1 -17966.423,E2 -17966.423} C_VEL
LIN {X 0,Y 279.538,Z 486.405,A -85,B 0,C 180,E1 -17967.763,E2 -17967.763} C_VEL
LIN {X 0,Y 278.65,Z 484.97,A -85,B 0,C 180,E1 -17968.125,E2 -17968.125} C_VEL
LIN {X 0,Y 275.967,Z 482.394,A -85,B 0,C 180,E1 -17969.169,E2 -17969.169} C_VEL
LIN {X 0,Y 274.395,Z 479.714,A -85,B 0,C 180,E1 -17969.865,E2 -17969.865} C_VEL
LIN {X 0,Y 271.694,Z 477.526,A -85,B 0,C 180,E1 -17970.987,E2 -17970.987} C_VEL
LIN {X 0,Y 270.365,Z 474.791,A -85,B 0,C 180,E1 -17971.786,E2 -17971.786} C_VEL
LIN {X 0,Y 270.269,Z 474.074,A -85,B 0,C 180,E1 -17972.296,E2 -17972.296} C_VEL
LIN {X 0,Y 270.23,Z 474.022,A -85,B 0,C 180,E1 -17975.538,E2 -17975.538} C_VEL
LIN {X 0,Y 270.294,Z 474.048,A -85,B 0,C 180,E1 -17980.244,E2 -17980.244} C_VEL
LIN {X 0,Y 270.39,Z 474.034,A -85,B 0,C 180,E1 -17984.935,E2 -17984.935} C_VEL
LIN {X 0,Y 270.435,Z 474.025,A -85,B 0,C 180,E1 -17989.519,E2 -17989.519} C_VEL
LIN {X 0,Y 270.602,Z 474.008,A -85,B 0,C 180,E1 -17992.539,E2 -17992.539} C_VEL
LIN {X 0,Y 270.781,Z 473.98,A -85,B 0,C 180,E1 -17998.513,E2 -17998.513} C_VEL
LIN {X 0,Y 270.781,Z 474.004,A -85,B 0,C 180,E1 -18001.488,E2 -18001.488} C_VEL
LIN {X 0,Y 270.593,Z 474.009,A -85,B 0,C 180,E1 -18007.462,E2 -18007.462} C_VEL
LIN {X 0,Y 270.407,Z 474.045,A -85,B 0,C 180,E1 -18010.483,E2 -18010.483} C_VEL
LIN {X 0,Y 270.391,Z 474.045,A -85,B 0,C 180,E1 -18015.066,E2 -18015.066} C_VEL
LIN {X 0,Y 270.294,Z 473.98,A -85,B 0,C 180,E1 -18019.756,E2 -18019.756} C_VEL
LIN {X 0,Y 270.271,Z 474.067,A -85,B 0,C 180,E1 -18024.586,E2 -18024.586} C_VEL
LIN {X 0,Y 270.309,Z 474.192,A -85,B 0,C 180,E1 -18027.484,E2 -18027.484} C_VEL
LIN {X 0,Y 270.549,Z 475.295,A -85,B 0,C 180,E1 -18028.003,E2 -18028.003} C_VEL
LIN {X 0,Y 271.964,Z 477.847,A -85,B 0,C 180,E1 -18028.717,E2 -18028.717} C_VEL
LIN {X 0,Y 274.734,Z 480.151,A -85,B 0,C 180,E1 -18029.864,E2 -18029.864} C_VEL
LIN {X 0,Y 276.584,Z 483.193,A -85,B 0,C 180,E1 -18030.67,E2 -18030.67} C_VEL
LIN {X 0,Y 279.03,Z 485.59,A -85,B 0,C 180,E1 -18031.615,E2 -18031.615} C_VEL
LIN {X 0,Y 279.971,Z 487.148,A -85,B 0,C 180,E1 -18031.998,E2 -18031.998} C_VEL
LIN {X 0,Y 281.245,Z 489.839,A -85,B 0,C 180,E1 -18032.532,E2 -18032.532} C_VEL
LIN {X 0,Y 282.61,Z 495.469,A -85,B 0,C 180,E1 -18033.215,E2 -18033.215} C_VEL
LIN {X 0,Y 283.93,Z 501.254,A -85,B 0,C 180,E1 -18033.873,E2 -18033.873} C_VEL
LIN {X 0,Y 285.166,Z 504.185,A -85,B 0,C 180,E1 -18034.366,E2 -18034.366} C_VEL
LIN {X 0,Y 289.218,Z 510.655,A -85,B 0,C 180,E1 -18035.783,E2 -18035.783} C_VEL
LIN {X 0,Y 294.685,Z 519.538,A -85,B 0,C 180,E1 -18037.569,E2 -18037.569} C_VEL
LIN {X 0,Y 302.018,Z 532.862,A -85,B 0,C 180,E1 -18039.815,E2 -18039.815} C_VEL
LIN {X 0,Y 308.896,Z 546.436,A -85,B 0,C 180,E1 -18041.775,E2 -18041.775} C_VEL
LIN {X 0,Y 314.738,Z 559.387,A -85,B 0,C 180,E1 -18043.365,E2 -18043.365} C_VEL
LIN {X 0,Y 309.09,Z 666.598,A -85,B 0,C 180,E1 -18045.753,E2 -18045.753} C_VEL
LIN {X 0,Y 307.488,Z 692.393,A -85,B 0,C 180,E1 -18046.373,E2 -18046.373} C_VEL
LIN {X 0,Y 305.269,Z 711.01,A -85,B 0,C 180,E1 -18047.055,E2 -18047.055} C_VEL
LIN {X 0,Y 303.089,Z 724.646,A -85,B 0,C 180,E1 -18047.745,E2 -18047.745} C_VEL
LIN {X 0,Y 300.672,Z 737.561,A -85,B 0,C 180,E1 -18048.577,E2 -18048.577} C_VEL
LIN {X 0,Y 297.893,Z 750.084,A -85,B 0,C 180,E1 -18049.551,E2 -18049.551} C_VEL
LIN {X 0,Y 294.987,Z 761.722,A -85,B 0,C 180,E1 -18050.63,E2 -18050.63} C_VEL
LIN {X 0,Y 291.441,Z 774.548,A -85,B 0,C 180,E1 -18052.055,E2 -18052.055} C_VEL
LIN {X 0,Y 288.442,Z 784.542,A -85,B 0,C 180,E1 -18053.35,E2 -18053.35} C_VEL
LIN {X 0,Y 284.916,Z 795.513,A -85,B 0,C 180,E1 -18055.006,E2 -18055.006} C_VEL
LIN {X 0,Y 281.566,Z 805.2,A -85,B 0,C 180,E1 -18056.694,E2 -18056.694} C_VEL
LIN {X 0,Y 277.947,Z 815.406,A -85,B 0,C 180,E1 -18058.779,E2 -18058.779} C_VEL
LIN {X 0,Y 274.794,Z 824.368,A -85,B 0,C 180,E1 -18060.927,E2 -18060.927} C_VEL
LIN {X 0,Y 271.844,Z 832.257,A -85,B 0,C 180,E1 -18063.101,E2 -18063.101} C_VEL
LIN {X 0,Y 269.342,Z 839.223,A -85,B 0,C 180,E1 -18065.324,E2 -18065.324} C_VEL
LIN {X 0,Y 267.226,Z 845.366,A -85,B 0,C 180,E1 -18067.583,E2 -18067.583} C_VEL
LIN {X 0,Y 264.952,Z 852.318,A -85,B 0,C 180,E1 -18070.636,E2 -18070.636} C_VEL
LIN {X 0,Y 263.642,Z 856.792,A -85,B 0,C 180,E1 -18072.949,E2 -18072.949} C_VEL
LIN {X 0,Y 262.337,Z 861.697,A -85,B 0,C 180,E1 -18076.048,E2 -18076.048} C_VEL
LIN {X 0,Y 261.459,Z 865.552,A -85,B 0,C 180,E1 -18079.155,E2 -18079.155} C_VEL
LIN {X 0,Y 261.133,Z 868.411,A -85,B 0,C 180,E1 -18082.267,E2 -18082.267} C_VEL
LIN {X 0,Y 261.046,Z 870.302,A -85,B 0,C 180,E1 -18085.367,E2 -18085.367} C_VEL
LIN {X 0,Y 261.046,Z 870.98,A -85,B 0,C 180,E1 -18086.913,E2 -18086.913} C_VEL
LIN {X 0,Y 261.092,Z 871.456,A -85,B 0,C 180,E1 -18090,E2 -18090} C_VEL
LIN {X 0,Y 261.046,Z 870.98,A -85,B 0,C 180,E1 -18093.087,E2 -18093.087} C_VEL
LIN {X 0,Y 261.045,Z 869.55,A -85,B 0,C 180,E1 -18096.182,E2 -18096.182} C_VEL
LIN {X 0,Y 261.262,Z 867.158,A -85,B 0,C 180,E1 -18099.288,E2 -18099.288} C_VEL
LIN {X 0,Y 262.076,Z 862.738,A -85,B 0,C 180,E1 -18103.176,E2 -18103.176} C_VEL
LIN {X 0,Y 263.094,Z 858.682,A -85,B 0,C 180,E1 -18105.916,E2 -18105.916} C_VEL
LIN {X 0,Y 264.485,Z 853.863,A -85,B 0,C 180,E1 -18108.594,E2 -18108.594} C_VEL
LIN {X 0,Y 266.05,Z 849.002,A -85,B 0,C 180,E1 -18110.892,E2 -18110.892} C_VEL
LIN {X 0,Y 268.541,Z 841.498,A -85,B 0,C 180,E1 -18113.866,E2 -18113.866} C_VEL
LIN {X 0,Y 270.97,Z 834.675,A -85,B 0,C 180,E1 -18116.162,E2 -18116.162} C_VEL
LIN {X 0,Y 273.84,Z 827.127,A -85,B 0,C 180,E1 -18118.345,E2 -18118.345} C_VEL
LIN {X 0,Y 276.867,Z 818.54,A -85,B 0,C 180,E1 -18120.509,E2 -18120.509} C_VEL
LIN {X 0,Y 280.296,Z 808.75,A -85,B 0,C 180,E1 -18122.62,E2 -18122.62} C_VEL
LIN {X 0,Y 283.838,Z 798.53,A -85,B 0,C 180,E1 -18124.499,E2 -18124.499} C_VEL
LIN {X 0,Y 286.978,Z 789.111,A -85,B 0,C 180,E1 -18125.997,E2 -18125.997} C_VEL
LIN {X 0,Y 290.622,Z 777.156,A -85,B 0,C 180,E1 -18127.633,E2 -18127.633} C_VEL
LIN {X 0,Y 293.731,Z 766.219,A -85,B 0,C 180,E1 -18128.907,E2 -18128.907} C_VEL
LIN {X 0,Y 297.028,Z 753.566,A -85,B 0,C 180,E1 -18130.147,E2 -18130.147} C_VEL
LIN {X 0,Y 299.583,Z 742.578,A -85,B 0,C 180,E1 -18131.06,E2 -18131.06} C_VEL
LIN {X 0,Y 302.148,Z 729.824,A -85,B 0,C 180,E1 -18131.946,E2 -18131.946} C_VEL
LIN {X 0,Y 304.475,Z 716.374,A -85,B 0,C 180,E1 -18132.69,E2 -18132.69} C_VEL
LIN {X 0,Y 306.344,Z 703.006,A -85,B 0,C 180,E1 -18133.264,E2 -18133.264} C_VEL
LIN {X 0,Y 307.698,Z 689.553,A -85,B 0,C 180,E1 -18133.702,E2 -18133.702} C_VEL
LIN {X 0,Y 309.839,Z 652.268,A -85,B 0,C 180,E1 -18134.566,E2 -18134.566} C_VEL
LIN {X 0,Y 314.735,Z 559.42,A -85,B 0,C 180,E1 -18136.634,E2 -18136.634} C_VEL
LIN {X 0,Y 307.859,Z 544.357,A -85,B 0,C 180,E1 -18138.511,E2 -18138.511} C_VEL
LIN {X 0,Y 300.154,Z 529.335,A -85,B 0,C 180,E1 -18140.741,E2 -18140.741} C_VEL
LIN {X 0,Y 293.306,Z 517.211,A -85,B 0,C 180,E1 -18142.871,E2 -18142.871} C_VEL
LIN {X 0,Y 286.364,Z 506.072,A -85,B 0,C 180,E1 -18145.207,E2 -18145.207} C_VEL
LIN {X 0,Y 283.244,Z 501.299,A -85,B 0,C 180,E1 -18146.33,E2 -18146.33} C_VEL
LIN {X 0,Y 279.746,Z 496.142,A -85,B 0,C 180,E1 -18147.653,E2 -18147.653} C_VEL
LIN {X 0,Y 275.934,Z 491.08,A -85,B 0,C 180,E1 -18149.164,E2 -18149.164} C_VEL
LIN {X 0,Y 273.182,Z 487.969,A -85,B 0,C 180,E1 -18150.297,E2 -18150.297} C_VEL
LIN {X 0,Y 271.845,Z 485.928,A -85,B 0,C 180,E1 -18150.898,E2 -18150.898} C_VEL
LIN {X 0,Y 269.25,Z 483.493,A -85,B 0,C 180,E1 -18152.032,E2 -18152.032} C_VEL
LIN {X 0,Y 267.604,Z 480.618,A -85,B 0,C 180,E1 -18152.861,E2 -18152.861} C_VEL
LIN {X 0,Y 264.877,Z 478.672,A -85,B 0,C 180,E1 -18154.142,E2 -18154.142} C_VEL
LIN {X 0,Y 263.504,Z 476.281,A -85,B 0,C 180,E1 -18154.939,E2 -18154.939} C_VEL
LIN {X 0,Y 263.25,Z 475.071,A -85,B 0,C 180,E1 -18155.608,E2 -18155.608} C_VEL
LIN {X 0,Y 263.257,Z 474.854,A -85,B 0,C 180,E1 -18159.693,E2 -18159.693} C_VEL
LIN {X 0,Y 263.339,Z 474.93,A -85,B 0,C 180,E1 -18164.521,E2 -18164.521} C_VEL
LIN {X 0,Y 263.349,Z 474.93,A -85,B 0,C 180,E1 -18169.233,E2 -18169.233} C_VEL
LIN {X 0,Y 263.553,Z 474.885,A -85,B 0,C 180,E1 -18172.338,E2 -18172.338} C_VEL
LIN {X 0,Y 263.745,Z 474.878,A -85,B 0,C 180,E1 -18178.473,E2 -18178.473} C_VEL
LIN {X 0,Y 263.745,Z 474.854,A -85,B 0,C 180,E1 -18181.527,E2 -18181.527} C_VEL
LIN {X 0,Y 263.564,Z 474.884,A -85,B 0,C 180,E1 -18187.661,E2 -18187.661} C_VEL
LIN {X 0,Y 263.368,Z 474.902,A -85,B 0,C 180,E1 -18190.765,E2 -18190.765} C_VEL
LIN {X 0,Y 263.338,Z 474.91,A -85,B 0,C 180,E1 -18195.478,E2 -18195.478} C_VEL
LIN {X 0,Y 263.257,Z 474.922,A -85,B 0,C 180,E1 -18200.307,E2 -18200.307} C_VEL
LIN {X 0,Y 263.225,Z 475.099,A -85,B 0,C 180,E1 -18204.802,E2 -18204.802} C_VEL
LIN {X 0,Y 263.501,Z 476.269,A -85,B 0,C 180,E1 -18205.472,E2 -18205.472} C_VEL
LIN {X 0,Y 264.893,Z 478.633,A -85,B 0,C 180,E1 -18206.279,E2 -18206.279} C_VEL
LIN {X 0,Y 267.883,Z 481.054,A -85,B 0,C 180,E1 -18207.695,E2 -18207.695} C_VEL
LIN {X 0,Y 269.723,Z 484.122,A -85,B 0,C 180,E1 -18208.606,E2 -18208.606} C_VEL
LIN {X 0,Y 272.382,Z 486.625,A -85,B 0,C 180,E1 -18209.755,E2 -18209.755} C_VEL
LIN {X 0,Y 274.725,Z 489.929,A -85,B 0,C 180,E1 -18210.772,E2 -18210.772} C_VEL
LIN {X 0,Y 276.638,Z 491.877,A -85,B 0,C 180,E1 -18211.532,E2 -18211.532} C_VEL
LIN {X 0,Y 279.428,Z 495.55,A -85,B 0,C 180,E1 -18212.633,E2 -18212.633} C_VEL
LIN {X 0,Y 281.002,Z 497.536,A -85,B 0,C 180,E1 -18213.226,E2 -18213.226} C_VEL
LIN {X 0,Y 284.756,Z 502.451,A -85,B 0,C 180,E1 -18214.586,E2 -18214.586} C_VEL
LIN {X 0,Y 292.057,Z 511.269,A -85,B 0,C 180,E1 -18216.984,E2 -18216.984} C_VEL
LIN {X 0,Y 298.298,Z 517.718,A -85,B 0,C 180,E1 -18218.832,E2 -18218.832} C_VEL
LIN {X 0,Y 304.563,Z 523.9,A -85,B 0,C 180,E1 -18220.764,E2 -18220.764} C_VEL
LIN {X 0,Y 307.818,Z 526.876,A -85,B 0,C 180,E1 -18221.81,E2 -18221.81} C_VEL
LIN {X 0,Y 312.539,Z 531.255,A -85,B 0,C 180,E1 -18223.428,E2 -18223.428} C_VEL
LIN {X 0,Y 317.81,Z 536.51,A -85,B 0,C 180,E1 -18225.386,E2 -18225.386} C_VEL
LIN {X 0,Y 320.574,Z 539.141,A -85,B 0,C 180,E1 -18226.48,E2 -18226.48} C_VEL
LIN {X 0,Y 324.798,Z 543.351,A -85,B 0,C 180,E1 -18228.22,E2 -18228.22} C_VEL
LIN {X 0,Y 326.731,Z 545.192,A -85,B 0,C 180,E1 -18229.024,E2 -18229.024} C_VEL
LIN {X 0,Y 330.942,Z 549.411,A -85,B 0,C 180,E1 -18230.83,E2 -18230.83} C_VEL
LIN {X 0,Y 333.369,Z 551.525,A -85,B 0,C 180,E1 -18231.869,E2 -18231.869} C_VEL
LIN {X 0,Y 337.404,Z 555.638,A -85,B 0,C 180,E1 -18233.691,E2 -18233.691} C_VEL
LIN {X 0,Y 340.477,Z 558.274,A -85,B 0,C 180,E1 -18235.094,E2 -18235.094} C_VEL
LIN {X 0,Y 344.676,Z 562.391,A -85,B 0,C 180,E1 -18237.103,E2 -18237.103} C_VEL
LIN {X 0,Y 347.855,Z 564.95,A -85,B 0,C 180,E1 -18238.653,E2 -18238.653} C_VEL
LIN {X 0,Y 351.399,Z 568.486,A -85,B 0,C 180,E1 -18240.518,E2 -18240.518} C_VEL
LIN {X 0,Y 355.235,Z 571.597,A -85,B 0,C 180,E1 -18242.591,E2 -18242.591} C_VEL
LIN {X 0,Y 358.658,Z 575.183,A -85,B 0,C 180,E1 -18244.622,E2 -18244.622} C_VEL
LIN {X 0,Y 362.001,Z 577.521,A -85,B 0,C 180,E1 -18246.662,E2 -18246.662} C_VEL
LIN {X 0,Y 363.251,Z 578.59,A -85,B 0,C 180,E1 -18247.483,E2 -18247.483} C_VEL
LIN {X 0,Y 365.883,Z 581.421,A -85,B 0,C 180,E1 -18249.352,E2 -18249.352} C_VEL
LIN {X 0,Y 369.176,Z 583.939,A -85,B 0,C 180,E1 -18251.828,E2 -18251.828} C_VEL
LIN {X 0,Y 371.501,Z 585.315,A -85,B 0,C 180,E1 -18253.749,E2 -18253.749} C_VEL
LIN {X 0,Y 373.706,Z 588.039,A -85,B 0,C 180,E1 -18255.968,E2 -18255.968} C_VEL
LIN {X 0,Y 376.005,Z 590.036,A -85,B 0,C 180,E1 -18258.604,E2 -18258.604} C_VEL
LIN {X 0,Y 377.873,Z 590.994,A -85,B 0,C 180,E1 -18261.132,E2 -18261.132} C_VEL
LIN {X 0,Y 379.229,Z 591.686,A -85,B 0,C 180,E1 -18263.616,E2 -18263.616} C_VEL
LIN {X 0,Y 380.041,Z 592.268,A -85,B 0,C 180,E1 -18265.758,E2 -18265.758} C_VEL
LIN {X 0,Y 380.556,Z 592.43,A -85,B 0,C 180,E1 -18267.883,E2 -18267.883} C_VEL
LIN {X 0,Y 380.744,Z 592.489,A -85,B 0,C 180,E1 -18270,E2 -18270} C_VEL
LIN {X 0,Y 380.557,Z 592.428,A -85,B 0,C 180,E1 -18272.117,E2 -18272.117} C_VEL
LIN {X 0,Y 379.883,Z 592.134,A -85,B 0,C 180,E1 -18274.749,E2 -18274.749} C_VEL
LIN {X 0,Y 378.695,Z 591.428,A -85,B 0,C 180,E1 -18277.464,E2 -18277.464} C_VEL
LIN {X 0,Y 376.89,Z 590.562,A -85,B 0,C 180,E1 -18280.276,E2 -18280.276} C_VEL
LIN {X 0,Y 374.802,Z 589.053,A -85,B 0,C 180,E1 -18282.825,E2 -18282.825} C_VEL
LIN {X 0,Y 372.629,Z 586.797,A -85,B 0,C 180,E1 -18285.151,E2 -18285.151} C_VEL
LIN {X 0,Y 370.955,Z 584.856,A -85,B 0,C 180,E1 -18286.733,E2 -18286.733} C_VEL
LIN {X 0,Y 368.007,Z 583.148,A -85,B 0,C 180,E1 -18289.075,E2 -18289.075} C_VEL
LIN {X 0,Y 364.86,Z 580.44,A -85,B 0,C 180,E1 -18291.4,E2 -18291.4} C_VEL
LIN {X 0,Y 362.457,Z 577.846,A -85,B 0,C 180,E1 -18293.061,E2 -18293.061} C_VEL
LIN {X 0,Y 358.783,Z 575.287,A -85,B 0,C 180,E1 -18295.305,E2 -18295.305} C_VEL
LIN {X 0,Y 355.094,Z 571.478,A -85,B 0,C 180,E1 -18297.487,E2 -18297.487} C_VEL
LIN {X 0,Y 350.051,Z 567.306,A -85,B 0,C 180,E1 -18300.19,E2 -18300.19} C_VEL
LIN {X 0,Y 346.538,Z 563.756,A -85,B 0,C 180,E1 -18301.992,E2 -18301.992} C_VEL
LIN {X 0,Y 342.653,Z 560.529,A -85,B 0,C 180,E1 -18303.874,E2 -18303.874} C_VEL
LIN {X 0,Y 338.834,Z 556.737,A -85,B 0,C 180,E1 -18305.674,E2 -18305.674} C_VEL
LIN {X 0,Y 334.417,Z 552.755,A -85,B 0,C 180,E1 -18307.65,E2 -18307.65} C_VEL
LIN {X 0,Y 331.987,Z 550.224,A -85,B 0,C 180,E1 -18308.732,E2 -18308.732} C_VEL
LIN {X 0,Y 327.784,Z 546.368,A -85,B 0,C 180,E1 -18310.52,E2 -18310.52} C_VEL
LIN {X 0,Y 325.049,Z 543.523,A -85,B 0,C 180,E1 -18311.681,E2 -18311.681} C_VEL
LIN {X 0,Y 320.614,Z 539.217,A -85,B 0,C 180,E1 -18313.502,E2 -18313.502} C_VEL
LIN {X 0,Y 317.505,Z 536.241,A -85,B 0,C 180,E1 -18314.729,E2 -18314.729} C_VEL
LIN {X 0,Y 312.279,Z 531.038,A -85,B 0,C 180,E1 -18316.663,E2 -18316.663} C_VEL
LIN {X 0,Y 307.583,Z 526.653,A -85,B 0,C 180,E1 -18318.266,E2 -18318.266} C_VEL
LIN {X 0,Y 301.127,Z 520.618,A -85,B 0,C 180,E1 -18320.303,E2 -18320.303} C_VEL
LIN {X 0,Y 297.901,Z 517.351,A -85,B 0,C 180,E1 -18321.282,E2 -18321.282} C_VEL
LIN {X 0,Y 293.438,Z 512.646,A -85,B 0,C 180,E1 -18322.603,E2 -18322.603} C_VEL
LIN {X 0,Y 288.791,Z 507.507,A -85,B 0,C 180,E1 -18324.049,E2 -18324.049} C_VEL
LIN {X 0,Y 283.901,Z 501.134,A -85,B 0,C 180,E1 -18325.725,E2 -18325.725} C_VEL
LIN {X 0,Y 280.347,Z 496.512,A -85,B 0,C 180,E1 -18327.028,E2 -18327.028} C_VEL
LIN {X 0,Y 276.928,Z 492.386,A -85,B 0,C 180,E1 -18328.345,E2 -18328.345} C_VEL
LIN {X 0,Y 275.959,Z 491.029,A -85,B 0,C 180,E1 -18328.742,E2 -18328.742} C_VEL
LIN {X 0,Y 273.209,Z 488.05,A -85,B 0,C 180,E1 -18329.867,E2 -18329.867} C_VEL
LIN {X 0,Y 271.931,Z 486.028,A -85,B 0,C 180,E1 -18330.445,E2 -18330.445} C_VEL
LIN {X 0,Y 269.175,Z 483.421,A -85,B 0,C 180,E1 -18331.65,E2 -18331.65} C_VEL
LIN {X 0,Y 267.465,Z 480.544,A -85,B 0,C 180,E1 -18332.507,E2 -18332.507} C_VEL
LIN {X 0,Y 264.895,Z 478.614,A -85,B 0,C 180,E1 -18333.722,E2 -18333.722} C_VEL
LIN {X 0,Y 263.413,Z 476.005,A -85,B 0,C 180,E1 -18334.625,E2 -18334.625} C_VEL
LIN {X 0,Y 263.193,Z 474.996,A -85,B 0,C 180,E1 -18335.288,E2 -18335.288} C_VEL
LIN {X 0,Y 263.257,Z 474.922,A -85,B 0,C 180,E1 -18339.693,E2 -18339.693} C_VEL
LIN {X 0,Y 263.338,Z 474.909,A -85,B 0,C 180,E1 -18344.522,E2 -18344.522} C_VEL
LIN {X 0,Y 263.368,Z 474.903,A -85,B 0,C 180,E1 -18349.235,E2 -18349.235} C_VEL
LIN {X 0,Y 263.564,Z 474.886,A -85,B 0,C 180,E1 -18352.339,E2 -18352.339} C_VEL
LIN {X 0,Y 263.745,Z 474.856,A -85,B 0,C 180,E1 -18358.473,E2 -18358.473} C_VEL
LIN {X 0,Y 263.745,Z 474.88,A -85,B 0,C 180,E1 -18361.527,E2 -18361.527} C_VEL
LIN {X 0,Y 263.553,Z 474.883,A -85,B 0,C 180,E1 -18367.662,E2 -18367.662} C_VEL
LIN {X 0,Y 263.349,Z 474.929,A -85,B 0,C 180,E1 -18370.767,E2 -18370.767} C_VEL
LIN {X 0,Y 263.339,Z 474.93,A -85,B 0,C 180,E1 -18375.479,E2 -18375.479} C_VEL
LIN {X 0,Y 263.257,Z 474.854,A -85,B 0,C 180,E1 -18380.307,E2 -18380.307} C_VEL
LIN {X 0,Y 263.258,Z 475.151,A -85,B 0,C 180,E1 -18384.44,E2 -18384.44} C_VEL
LIN {X 0,Y 263.504,Z 476.264,A -85,B 0,C 180,E1 -18385.061,E2 -18385.061} C_VEL
LIN {X 0,Y 264.88,Z 478.642,A -85,B 0,C 180,E1 -18385.858,E2 -18385.858} C_VEL
LIN {X 0,Y 267.323,Z 480.47,A -85,B 0,C 180,E1 -18387.014,E2 -18387.014} C_VEL
LIN {X 0,Y 267.928,Z 481.067,A -85,B 0,C 180,E1 -18387.298,E2 -18387.298} C_VEL
LIN {X 0,Y 269.711,Z 484.093,A -85,B 0,C 180,E1 -18388.183,E2 -18388.183} C_VEL
LIN {X 0,Y 272.328,Z 486.448,A -85,B 0,C 180,E1 -18389.31,E2 -18389.31} C_VEL
LIN {X 0,Y 274.634,Z 489.863,A -85,B 0,C 180,E1 -18390.321,E2 -18390.321} C_VEL
LIN {X 0,Y 276.635,Z 491.979,A -85,B 0,C 180,E1 -18391.121,E2 -18391.121} C_VEL
LIN {X 0,Y 281.414,Z 498.562,A -85,B 0,C 180,E1 -18392.986,E2 -18392.986} C_VEL
LIN {X 0,Y 285.166,Z 504.185,A -85,B 0,C 180,E1 -18394.366,E2 -18394.366} C_VEL
LIN {X 0,Y 287.151,Z 508.31,A -85,B 0,C 180,E1 -18395.112,E2 -18395.112} C_VEL
LIN {X 0,Y 289.729,Z 516.279,A -85,B 0,C 180,E1 -18396.153,E2 -18396.153} C_VEL
LIN {X 0,Y 291.616,Z 522.987,A -85,B 0,C 180,E1 -18396.922,E2 -18396.922} C_VEL
LIN {X 0,Y 293.861,Z 529.368,A -85,B 0,C 180,E1 -18397.746,E2 -18397.746} C_VEL
LIN {X 0,Y 301.179,Z 543.396,A -85,B 0,C 180,E1 -18400.007,E2 -18400.007} C_VEL
LIN {X 0,Y 307.871,Z 557.638,A -85,B 0,C 180,E1 -18401.946,E2 -18401.946} C_VEL
LIN {X 0,Y 309.778,Z 562.117,A -85,B 0,C 180,E1 -18402.484,E2 -18402.484} C_VEL
LIN {X 0,Y 302.939,Z 685.249,A -85,B 0,C 180,E1 -18405.256,E2 -18405.256} C_VEL
LIN {X 0,Y 301.558,Z 699.798,A -85,B 0,C 180,E1 -18405.699,E2 -18405.699} C_VEL
LIN {X 0,Y 299.726,Z 713.097,A -85,B 0,C 180,E1 -18406.235,E2 -18406.235} C_VEL
LIN {X 0,Y 297.847,Z 724.435,A -85,B 0,C 180,E1 -18406.822,E2 -18406.822} C_VEL
LIN {X 0,Y 295.436,Z 736.983,A -85,B 0,C 180,E1 -18407.634,E2 -18407.634} C_VEL
LIN {X 0,Y 292.501,Z 749.874,A -85,B 0,C 180,E1 -18408.644,E2 -18408.644} C_VEL
LIN {X 0,Y 289.486,Z 761.51,A -85,B 0,C 180,E1 -18409.731,E2 -18409.731} C_VEL
LIN {X 0,Y 285.82,Z 774.336,A -85,B 0,C 180,E1 -18411.171,E2 -18411.171} C_VEL
LIN {X 0,Y 282.711,Z 784.329,A -85,B 0,C 180,E1 -18412.481,E2 -18412.481} C_VEL
LIN {X 0,Y 279.042,Z 795.391,A -85,B 0,C 180,E1 -18414.177,E2 -18414.177} C_VEL
LIN {X 0,Y 275.572,Z 804.987,A -85,B 0,C 180,E1 -18415.871,E2 -18415.871} C_VEL
LIN {X 0,Y 271.814,Z 815.194,A -85,B 0,C 180,E1 -18417.992,E2 -18417.992} C_VEL
LIN {X 0,Y 268.931,Z 823.018,A -85,B 0,C 180,E1 -18419.874,E2 -18419.874} C_VEL
LIN {X 0,Y 265.407,Z 832.043,A -85,B 0,C 180,E1 -18422.394,E2 -18422.394} C_VEL
LIN {X 0,Y 262.785,Z 839.009,A -85,B 0,C 180,E1 -18424.666,E2 -18424.666} C_VEL
LIN {X 0,Y 260.551,Z 845.152,A -85,B 0,C 180,E1 -18426.977,E2 -18426.977} C_VEL
LIN {X 0,Y 258.159,Z 852.104,A -85,B 0,C 180,E1 -18430.106,E2 -18430.106} C_VEL
LIN {X 0,Y 256.759,Z 856.579,A -85,B 0,C 180,E1 -18432.477,E2 -18432.477} C_VEL
LIN {X 0,Y 255.373,Z 861.485,A -85,B 0,C 180,E1 -18435.66,E2 -18435.66} C_VEL
LIN {X 0,Y 254.417,Z 865.34,A -85,B 0,C 180,E1 -18438.851,E2 -18438.851} C_VEL
LIN {X 0,Y 254.063,Z 868.2,A -85,B 0,C 180,E1 -18442.05,E2 -18442.05} C_VEL
LIN {X 0,Y 253.973,Z 870.092,A -85,B 0,C 180,E1 -18445.238,E2 -18445.238} C_VEL
LIN {X 0,Y 253.945,Z 870.77,A -85,B 0,C 180,E1 -18446.827,E2 -18446.827} C_VEL
LIN {X 0,Y 254.021,Z 871.247,A -85,B 0,C 180,E1 -18450,E2 -18450} C_VEL
LIN {X 0,Y 253.945,Z 870.77,A -85,B 0,C 180,E1 -18453.173,E2 -18453.173} C_VEL
LIN {X 0,Y 253.955,Z 869.339,A -85,B 0,C 180,E1 -18456.355,E2 -18456.355} C_VEL
LIN {X 0,Y 254.2,Z 866.946,A -85,B 0,C 180,E1 -18459.548,E2 -18459.548} C_VEL
LIN {X 0,Y 255.091,Z 862.526,A -85,B 0,C 180,E1 -18463.543,E2 -18463.543} C_VEL
LIN {X 0,Y 256.059,Z 858.841,A -85,B 0,C 180,E1 -18466.129,E2 -18466.129} C_VEL
LIN {X 0,Y 257.67,Z 853.651,A -85,B 0,C 180,E1 -18469.105,E2 -18469.105} C_VEL
LIN {X 0,Y 259.325,Z 848.789,A -85,B 0,C 180,E1 -18471.46,E2 -18471.46} C_VEL
LIN {X 0,Y 261.995,Z 841.118,A -85,B 0,C 180,E1 -18474.567,E2 -18474.567} C_VEL
LIN {X 0,Y 264.499,Z 834.462,A -85,B 0,C 180,E1 -18476.853,E2 -18476.853} C_VEL
LIN {X 0,Y 267.499,Z 826.914,A -85,B 0,C 180,E1 -18479.081,E2 -18479.081} C_VEL
LIN {X 0,Y 270.679,Z 818.327,A -85,B 0,C 180,E1 -18481.284,E2 -18481.284} C_VEL
LIN {X 0,Y 274.24,Z 808.536,A -85,B 0,C 180,E1 -18483.434,E2 -18483.434} C_VEL
LIN {X 0,Y 278.291,Z 797.311,A -85,B 0,C 180,E1 -18485.509,E2 -18485.509} C_VEL
LIN {X 0,Y 281.378,Z 788.333,A -85,B 0,C 180,E1 -18486.94,E2 -18486.94} C_VEL
LIN {X 0,Y 284.982,Z 776.945,A -85,B 0,C 180,E1 -18488.512,E2 -18488.512} C_VEL
LIN {X 0,Y 288.208,Z 766.008,A -85,B 0,C 180,E1 -18489.799,E2 -18489.799} C_VEL
LIN {X 0,Y 291.606,Z 753.355,A -85,B 0,C 180,E1 -18491.051,E2 -18491.051} C_VEL
LIN {X 0,Y 294.595,Z 740.722,A -85,B 0,C 180,E1 -18492.095,E2 -18492.095} C_VEL
LIN {X 0,Y 296.941,Z 729.344,A -85,B 0,C 180,E1 -18492.881,E2 -18492.881} C_VEL
LIN {X 0,Y 299.293,Z 716.164,A -85,B 0,C 180,E1 -18493.612,E2 -18493.612} C_VEL
LIN {X 0,Y 301.198,Z 702.796,A -85,B 0,C 180,E1 -18494.192,E2 -18494.192} C_VEL
LIN {X 0,Y 302.608,Z 689.344,A -85,B 0,C 180,E1 -18494.631,E2 -18494.631} C_VEL
LIN {X 0,Y 304.707,Z 653.849,A -85,B 0,C 180,E1 -18495.466,E2 -18495.466} C_VEL
LIN {X 0,Y 309.741,Z 562.712,A -85,B 0,C 180,E1 -18497.504,E2 -18497.504} C_VEL
LIN {X 0,Y 309.465,Z 561.281,A -85,B 0,C 180,E1 -18497.607,E2 -18497.607} C_VEL
LIN {X 0,Y 302.774,Z 546.722,A -85,B 0,C 180,E1 -18499.519,E2 -18499.519} C_VEL
LIN {X 0,Y 296.18,Z 533.714,A -85,B 0,C 180,E1 -18501.517,E2 -18501.517} C_VEL
LIN {X 0,Y 289.987,Z 522.584,A -85,B 0,C 180,E1 -18503.521,E2 -18503.521} C_VEL
LIN {X 0,Y 283.194,Z 511.453,A -85,B 0,C 180,E1 -18505.895,E2 -18505.895} C_VEL
LIN {X 0,Y 280.089,Z 506.646,A -85,B 0,C 180,E1 -18507.058,E2 -18507.058} C_VEL
LIN {X 0,Y 276.974,Z 501.94,A -85,B 0,C 180,E1 -18508.283,E2 -18508.283} C_VEL
LIN {X 0,Y 273.312,Z 497.124,A -85,B 0,C 180,E1 -18509.781,E2 -18509.781} C_VEL
LIN {X 0,Y 270.388,Z 493.503,A -85,B 0,C 180,E1 -18511.046,E2 -18511.046} C_VEL
LIN {X 0,Y 269.414,Z 492.183,A -85,B 0,C 180,E1 -18511.491,E2 -18511.491} C_VEL
LIN {X 0,Y 266.796,Z 489.383,A -85,B 0,C 180,E1 -18512.694,E2 -18512.694} C_VEL
LIN {X 0,Y 265.321,Z 487.056,A -85,B 0,C 180,E1 -18513.449,E2 -18513.449} C_VEL
LIN {X 0,Y 262.657,Z 484.815,A -85,B 0,C 180,E1 -18514.764,E2 -18514.764} C_VEL
LIN {X 0,Y 260.769,Z 481.645,A -85,B 0,C 180,E1 -18515.857,E2 -18515.857} C_VEL
LIN {X 0,Y 258.018,Z 479.823,A -85,B 0,C 180,E1 -18517.372,E2 -18517.372} C_VEL
LIN {X 0,Y 256.52,Z 477.388,A -85,B 0,C 180,E1 -18518.378,E2 -18518.378} C_VEL
LIN {X 0,Y 256.242,Z 476.378,A -85,B 0,C 180,E1 -18518.828,E2 -18518.828} C_VEL
LIN {X 0,Y 256.219,Z 475.813,A -85,B 0,C 180,E1 -18519.529,E2 -18519.529} C_VEL
LIN {X 0,Y 256.275,Z 475.806,A -85,B 0,C 180,E1 -18524.083,E2 -18524.083} C_VEL
LIN {X 0,Y 256.288,Z 475.787,A -85,B 0,C 180,E1 -18527.327,E2 -18527.327} C_VEL
LIN {X 0,Y 256.51,Z 475.76,A -85,B 0,C 180,E1 -18532.126,E2 -18532.126} C_VEL
LIN {X 0,Y 256.493,Z 475.761,A -85,B 0,C 180,E1 -18536.858,E2 -18536.858} C_VEL
LIN {X 0,Y 256.752,Z 475.735,A -85,B 0,C 180,E1 -18540,E2 -18540} C_VEL
LIN {X 0,Y 256.494,Z 475.77,A -85,B 0,C 180,E1 -18543.141,E2 -18543.141} C_VEL
LIN {X 0,Y 256.532,Z 475.762,A -85,B 0,C 180,E1 -18547.873,E2 -18547.873} C_VEL
LIN {X 0,Y 256.304,Z 475.781,A -85,B 0,C 180,E1 -18551.066,E2 -18551.066} C_VEL
LIN {X 0,Y 256.274,Z 475.789,A -85,B 0,C 180,E1 -18555.916,E2 -18555.916} C_VEL
LIN {X 0,Y 256.188,Z 475.839,A -85,B 0,C 180,E1 -18560.893,E2 -18560.893} C_VEL
LIN {X 0,Y 256.27,Z 476.716,A -85,B 0,C 180,E1 -18561.746,E2 -18561.746} C_VEL
LIN {X 0,Y 257.72,Z 479.548,A -85,B 0,C 180,E1 -18562.867,E2 -18562.867} C_VEL
LIN {X 0,Y 260.433,Z 481.51,A -85,B 0,C 180,E1 -18564.385,E2 -18564.385} C_VEL
LIN {X 0,Y 261.365,Z 482.604,A -85,B 0,C 180,E1 -18564.907,E2 -18564.907} C_VEL
LIN {X 0,Y 263.19,Z 485.376,A -85,B 0,C 180,E1 -18565.929,E2 -18565.929} C_VEL
LIN {X 0,Y 265.667,Z 487.474,A -85,B 0,C 180,E1 -18567.139,E2 -18567.139} C_VEL
LIN {X 0,Y 267.954,Z 490.886,A -85,B 0,C 180,E1 -18568.277,E2 -18568.277} C_VEL
LIN {X 0,Y 270.045,Z 492.905,A -85,B 0,C 180,E1 -18569.207,E2 -18569.207} C_VEL
LIN {X 0,Y 272.728,Z 496.53,A -85,B 0,C 180,E1 -18570.395,E2 -18570.395} C_VEL
LIN {X 0,Y 274.296,Z 498.257,A -85,B 0,C 180,E1 -18571.04,E2 -18571.04} C_VEL
LIN {X 0,Y 277.369,Z 502.132,A -85,B 0,C 180,E1 -18572.273,E2 -18572.273} C_VEL
LIN {X 0,Y 282.373,Z 508.926,A -85,B 0,C 180,E1 -18574.163,E2 -18574.163} C_VEL
LIN {X 0,Y 289.6,Z 517.622,A -85,B 0,C 180,E1 -18576.589,E2 -18576.589} C_VEL
LIN {X 0,Y 295.745,Z 524.01,A -85,B 0,C 180,E1 -18578.432,E2 -18578.432} C_VEL
LIN {X 0,Y 302.291,Z 530.347,A -85,B 0,C 180,E1 -18580.402,E2 -18580.402} C_VEL
LIN {X 0,Y 305.755,Z 533.543,A -85,B 0,C 180,E1 -18581.506,E2 -18581.506} C_VEL
LIN {X 0,Y 310.78,Z 538.024,A -85,B 0,C 180,E1 -18583.182,E2 -18583.182} C_VEL
LIN {X 0,Y 316.037,Z 543.209,A -85,B 0,C 180,E1 -18585.108,E2 -18585.108} C_VEL
LIN {X 0,Y 318.937,Z 546.033,A -85,B 0,C 180,E1 -18586.238,E2 -18586.238} C_VEL
LIN {X 0,Y 323.43,Z 550.305,A -85,B 0,C 180,E1 -18588.068,E2 -18588.068} C_VEL
LIN {X 0,Y 329.072,Z 555.921,A -85,B 0,C 180,E1 -18590.443,E2 -18590.443} C_VEL
LIN {X 0,Y 331.786,Z 558.319,A -85,B 0,C 180,E1 -18591.604,E2 -18591.604} C_VEL
LIN {X 0,Y 336.065,Z 562.561,A -85,B 0,C 180,E1 -18593.52,E2 -18593.52} C_VEL
LIN {X 0,Y 339.031,Z 565.132,A -85,B 0,C 180,E1 -18594.865,E2 -18594.865} C_VEL
LIN {X 0,Y 343.283,Z 569.237,A -85,B 0,C 180,E1 -18596.897,E2 -18596.897} C_VEL
LIN {X 0,Y 346.538,Z 571.878,A -85,B 0,C 180,E1 -18598.477,E2 -18598.477} C_VEL
LIN {X 0,Y 350.143,Z 575.401,A -85,B 0,C 180,E1 -18600.345,E2 -18600.345} C_VEL
LIN {X 0,Y 353.909,Z 578.466,A -85,B 0,C 180,E1 -18602.374,E2 -18602.374} C_VEL
LIN {X 0,Y 357.767,Z 582.372,A -85,B 0,C 180,E1 -18604.637,E2 -18604.637} C_VEL
LIN {X 0,Y 361.959,Z 585.37,A -85,B 0,C 180,E1 -18607.213,E2 -18607.213} C_VEL
LIN {X 0,Y 364.899,Z 588.486,A -85,B 0,C 180,E1 -18609.293,E2 -18609.293} C_VEL
LIN {X 0,Y 368.229,Z 590.974,A -85,B 0,C 180,E1 -18611.78,E2 -18611.78} C_VEL
LIN {X 0,Y 370.435,Z 592.271,A -85,B 0,C 180,E1 -18613.584,E2 -18613.584} C_VEL
LIN {X 0,Y 372.792,Z 595.094,A -85,B 0,C 180,E1 -18615.933,E2 -18615.933} C_VEL
LIN {X 0,Y 375.109,Z 597.082,A -85,B 0,C 180,E1 -18618.576,E2 -18618.576} C_VEL
LIN {X 0,Y 376.998,Z 598.034,A -85,B 0,C 180,E1 -18621.12,E2 -18621.12} C_VEL
LIN {X 0,Y 378.502,Z 598.828,A -85,B 0,C 180,E1 -18623.953,E2 -18623.953} C_VEL
LIN {X 0,Y 379.173,Z 599.289,A -85,B 0,C 180,E1 -18625.748,E2 -18625.748} C_VEL
LIN {X 0,Y 379.722,Z 599.47,A -85,B 0,C 180,E1 -18628.076,E2 -18628.076} C_VEL
LIN {X 0,Y 379.879,Z 599.535,A -85,B 0,C 180,E1 -18630,E2 -18630} C_VEL
LIN {X 0,Y 379.692,Z 599.466,A -85,B 0,C 180,E1 -18632.121,E2 -18632.121} C_VEL
LIN {X 0,Y 379.013,Z 599.176,A -85,B 0,C 180,E1 -18634.759,E2 -18634.759} C_VEL
LIN {X 0,Y 377.818,Z 598.473,A -85,B 0,C 180,E1 -18637.482,E2 -18637.482} C_VEL
LIN {X 0,Y 376.003,Z 597.606,A -85,B 0,C 180,E1 -18640.301,E2 -18640.301} C_VEL
LIN {X 0,Y 373.895,Z 596.103,A -85,B 0,C 180,E1 -18642.856,E2 -18642.856} C_VEL
LIN {X 0,Y 371.699,Z 593.886,A -85,B 0,C 180,E1 -18645.19,E2 -18645.19} C_VEL
LIN {X 0,Y 370.022,Z 591.88,A -85,B 0,C 180,E1 -18646.777,E2 -18646.777} C_VEL
LIN {X 0,Y 367.045,Z 590.186,A -85,B 0,C 180,E1 -18649.127,E2 -18649.127} C_VEL
LIN {X 0,Y 363.768,Z 587.426,A -85,B 0,C 180,E1 -18651.535,E2 -18651.535} C_VEL
LIN {X 0,Y 361.216,Z 584.739,A -85,B 0,C 180,E1 -18653.263,E2 -18653.263} C_VEL
LIN {X 0,Y 357.327,Z 581.955,A -85,B 0,C 180,E1 -18655.638,E2 -18655.638} C_VEL
LIN {X 0,Y 353.553,Z 578.082,A -85,B 0,C 180,E1 -18657.83,E2 -18657.83} C_VEL
LIN {X 0,Y 348.865,Z 574.335,A -85,B 0,C 180,E1 -18660.312,E2 -18660.312} C_VEL
LIN {X 0,Y 345.243,Z 570.666,A -85,B 0,C 180,E1 -18662.167,E2 -18662.167} C_VEL
LIN {X 0,Y 340.943,Z 567.09,A -85,B 0,C 180,E1 -18664.229,E2 -18664.229} C_VEL
LIN {X 0,Y 337.131,Z 563.392,A -85,B 0,C 180,E1 -18666.003,E2 -18666.003} C_VEL
LIN {X 0,Y 332.497,Z 559.163,A -85,B 0,C 180,E1 -18668.071,E2 -18668.071} C_VEL
LIN {X 0,Y 330.296,Z 556.881,A -85,B 0,C 180,E1 -18669.032,E2 -18669.032} C_VEL
LIN {X 0,Y 325.973,Z 552.956,A -85,B 0,C 180,E1 -18670.866,E2 -18670.866} C_VEL
LIN {X 0,Y 323.187,Z 550.13,A -85,B 0,C 180,E1 -18672.029,E2 -18672.029} C_VEL
LIN {X 0,Y 318.503,Z 545.544,A -85,B 0,C 180,E1 -18673.937,E2 -18673.937} C_VEL
LIN {X 0,Y 312.763,Z 540.101,A -85,B 0,C 180,E1 -18676.094,E2 -18676.094} C_VEL
LIN {X 0,Y 310.076,Z 537.495,A -85,B 0,C 180,E1 -18677.048,E2 -18677.048} C_VEL
LIN {X 0,Y 305.389,Z 533.168,A -85,B 0,C 180,E1 -18678.611,E2 -18678.611} C_VEL
LIN {X 0,Y 298.56,Z 526.836,A -85,B 0,C 180,E1 -18680.734,E2 -18680.734} C_VEL
LIN {X 0,Y 294.36,Z 522.736,A -85,B 0,C 180,E1 -18681.972,E2 -18681.972} C_VEL
LIN {X 0,Y 285.902,Z 513.328,A -85,B 0,C 180,E1 -18684.612,E2 -18684.612} C_VEL
LIN {X 0,Y 276.912,Z 501.661,A -85,B 0,C 180,E1 -18687.901,E2 -18687.901} C_VEL
LIN {X 0,Y 273.322,Z 497.079,A -85,B 0,C 180,E1 -18689.364,E2 -18689.364} C_VEL
LIN {X 0,Y 270.495,Z 493.692,A -85,B 0,C 180,E1 -18690.58,E2 -18690.58} C_VEL
LIN {X 0,Y 269.478,Z 492.251,A -85,B 0,C 180,E1 -18691.046,E2 -18691.046} C_VEL
LIN {X 0,Y 266.765,Z 489.389,A -85,B 0,C 180,E1 -18692.291,E2 -18692.291} C_VEL
LIN {X 0,Y 265.449,Z 487.116,A -85,B 0,C 180,E1 -18692.975,E2 -18692.975} C_VEL
LIN {X 0,Y 262.771,Z 484.87,A -85,B 0,C 180,E1 -18694.293,E2 -18694.293} C_VEL
LIN {X 0,Y 260.691,Z 481.586,A -85,B 0,C 180,E1 -18695.484,E2 -18695.484} C_VEL
LIN {X 0,Y 257.871,Z 479.716,A -85,B 0,C 180,E1 -18697.042,E2 -18697.042} C_VEL
LIN {X 0,Y 256.45,Z 477.32,A -85,B 0,C 180,E1 -18698.011,E2 -18698.011} C_VEL
LIN {X 0,Y 256.182,Z 476.148,A -85,B 0,C 180,E1 -18698.66,E2 -18698.66} C_VEL
LIN {X 0,Y 256.175,Z 475.856,A -85,B 0,C 180,E1 -18699.106,E2 -18699.106} C_VEL
LIN {X 0,Y 256.274,Z 475.788,A -85,B 0,C 180,E1 -18704.084,E2 -18704.084} C_VEL
LIN {X 0,Y 256.304,Z 475.782,A -85,B 0,C 180,E1 -18708.934,E2 -18708.934} C_VEL
LIN {X 0,Y 256.532,Z 475.764,A -85,B 0,C 180,E1 -18712.127,E2 -18712.127} C_VEL
LIN {X 0,Y 256.709,Z 475.733,A -85,B 0,C 180,E1 -18718.432,E2 -18718.432} C_VEL
LIN {X 0,Y 256.708,Z 475.754,A -85,B 0,C 180,E1 -18721.569,E2 -18721.569} C_VEL
LIN {X 0,Y 256.476,Z 475.786,A -85,B 0,C 180,E1 -18726.293,E2 -18726.293} C_VEL
LIN {X 0,Y 256.422,Z 475.771,A -85,B 0,C 180,E1 -18729.465,E2 -18729.465} C_VEL
LIN {X 0,Y 256.245,Z 475.795,A -85,B 0,C 180,E1 -18734.291,E2 -18734.291} C_VEL
LIN {X 0,Y 256.197,Z 475.763,A -85,B 0,C 180,E1 -18737.563,E2 -18737.563} C_VEL
LIN {X 0,Y 256.212,Z 475.989,A -85,B 0,C 180,E1 -18740.786,E2 -18740.786} C_VEL
LIN {X 0,Y 256.473,Z 477.204,A -85,B 0,C 180,E1 -18741.574,E2 -18741.574} C_VEL
LIN {X 0,Y 257.868,Z 479.641,A -85,B 0,C 180,E1 -18742.536,E2 -18742.536} C_VEL
LIN {X 0,Y 260.607,Z 481.574,A -85,B 0,C 180,E1 -18744.059,E2 -18744.059} C_VEL
LIN {X 0,Y 261.347,Z 482.598,A -85,B 0,C 180,E1 -18744.483,E2 -18744.483} C_VEL
LIN {X 0,Y 263.172,Z 485.408,A -85,B 0,C 180,E1 -18745.507,E2 -18745.507} C_VEL
LIN {X 0,Y 265.737,Z 487.543,A -85,B 0,C 180,E1 -18746.757,E2 -18746.757} C_VEL
LIN {X 0,Y 267.911,Z 490.826,A -85,B 0,C 180,E1 -18747.841,E2 -18747.841} C_VEL
LIN {X 0,Y 270.028,Z 492.876,A -85,B 0,C 180,E1 -18748.783,E2 -18748.783} C_VEL
LIN {X 0,Y 272.684,Z 496.491,A -85,B 0,C 180,E1 -18749.961,E2 -18749.961} C_VEL
LIN {X 0,Y 274.285,Z 498.345,A -85,B 0,C 180,E1 -18750.624,E2 -18750.624} C_VEL
LIN {X 0,Y 278.623,Z 504.362,A -85,B 0,C 180,E1 -18752.371,E2 -18752.371} C_VEL
LIN {X 0,Y 282.768,Z 510.783,A -85,B 0,C 180,E1 -18753.948,E2 -18753.948} C_VEL
LIN {X 0,Y 288.536,Z 520.111,A -85,B 0,C 180,E1 -18755.989,E2 -18755.989} C_VEL
LIN {X 0,Y 293.861,Z 529.368,A -85,B 0,C 180,E1 -18757.746,E2 -18757.746} C_VEL
LIN {X 0,Y 296.001,Z 535.839,A -85,B 0,C 180,E1 -18758.52,E2 -18758.52} C_VEL
LIN {X 0,Y 300.161,Z 553.331,A -85,B 0,C 180,E1 -18760.138,E2 -18760.138} C_VEL
LIN {X 0,Y 301.34,Z 556.549,A -85,B 0,C 180,E1 -18760.516,E2 -18760.516} C_VEL
LIN {X 0,Y 304.838,Z 564.539,A -85,B 0,C 180,E1 -18761.552,E2 -18761.552} C_VEL
LIN {X 0,Y 298.959,Z 667.968,A -85,B 0,C 180,E1 -18763.891,E2 -18763.891} C_VEL
LIN {X 0,Y 297.362,Z 691.973,A -85,B 0,C 180,E1 -18764.484,E2 -18764.484} C_VEL
LIN {X 0,Y 295.039,Z 710.591,A -85,B 0,C 180,E1 -18765.177,E2 -18765.177} C_VEL
LIN {X 0,Y 292.694,Z 724.224,A -85,B 0,C 180,E1 -18765.868,E2 -18765.868} C_VEL
LIN {X 0,Y 289.988,Z 737.776,A -85,B 0,C 180,E1 -18766.761,E2 -18766.761} C_VEL
LIN {X 0,Y 287.185,Z 749.663,A -85,B 0,C 180,E1 -18767.704,E2 -18767.704} C_VEL
LIN {X 0,Y 284.072,Z 761.299,A -85,B 0,C 180,E1 -18768.8,E2 -18768.8} C_VEL
LIN {X 0,Y 280.284,Z 774.125,A -85,B 0,C 180,E1 -18770.254,E2 -18770.254} C_VEL
LIN {X 0,Y 277.041,Z 784.112,A -85,B 0,C 180,E1 -18771.574,E2 -18771.574} C_VEL
LIN {X 0,Y 273.185,Z 795.371,A -85,B 0,C 180,E1 -18773.329,E2 -18773.329} C_VEL
LIN {X 0,Y 269.64,Z 804.774,A -85,B 0,C 180,E1 -18775.012,E2 -18775.012} C_VEL
LIN {X 0,Y 265.72,Z 814.98,A -85,B 0,C 180,E1 -18777.167,E2 -18777.167} C_VEL
LIN {X 0,Y 262.25,Z 823.941,A -85,B 0,C 180,E1 -18779.392,E2 -18779.392} C_VEL
LIN {X 0,Y 259.032,Z 831.83,A -85,B 0,C 180,E1 -18781.654,E2 -18781.654} C_VEL
LIN {X 0,Y 256.268,Z 838.795,A -85,B 0,C 180,E1 -18783.974,E2 -18783.974} C_VEL
LIN {X 0,Y 253.848,Z 845.097,A -85,B 0,C 180,E1 -18786.407,E2 -18786.407} C_VEL
LIN {X 0,Y 251.371,Z 851.891,A -85,B 0,C 180,E1 -18789.545,E2 -18789.545} C_VEL
LIN {X 0,Y 249.882,Z 856.366,A -85,B 0,C 180,E1 -18791.979,E2 -18791.979} C_VEL
LIN {X 0,Y 248.424,Z 861.273,A -85,B 0,C 180,E1 -18795.25,E2 -18795.25} C_VEL
LIN {X 0,Y 247.381,Z 865.128,A -85,B 0,C 180,E1 -18798.53,E2 -18798.53} C_VEL
LIN {X 0,Y 246.983,Z 867.989,A -85,B 0,C 180,E1 -18801.821,E2 -18801.821} C_VEL
LIN {X 0,Y 246.882,Z 869.882,A -85,B 0,C 180,E1 -18805.101,E2 -18805.101} C_VEL
LIN {X 0,Y 246.849,Z 870.56,A -85,B 0,C 180,E1 -18806.736,E2 -18806.736} C_VEL
LIN {X 0,Y 246.952,Z 871.038,A -85,B 0,C 180,E1 -18810,E2 -18810} C_VEL
LIN {X 0,Y 246.849,Z 870.56,A -85,B 0,C 180,E1 -18813.264,E2 -18813.264} C_VEL
LIN {X 0,Y 246.869,Z 869.128,A -85,B 0,C 180,E1 -18816.539,E2 -18816.539} C_VEL
LIN {X 0,Y 247.138,Z 866.735,A -85,B 0,C 180,E1 -18819.824,E2 -18819.824} C_VEL
LIN {X 0,Y 248.107,Z 862.313,A -85,B 0,C 180,E1 -18823.932,E2 -18823.932} C_VEL
LIN {X 0,Y 249.072,Z 858.942,A -85,B 0,C 180,E1 -18826.389,E2 -18826.389} C_VEL
LIN {X 0,Y 250.848,Z 853.437,A -85,B 0,C 180,E1 -18829.645,E2 -18829.645} C_VEL
LIN {X 0,Y 252.61,Z 848.575,A -85,B 0,C 180,E1 -18832.06,E2 -18832.06} C_VEL
LIN {X 0,Y 255.467,Z 840.903,A -85,B 0,C 180,E1 -18835.239,E2 -18835.239} C_VEL
LIN {X 0,Y 258.092,Z 834.249,A -85,B 0,C 180,E1 -18837.575,E2 -18837.575} C_VEL
LIN {X 0,Y 261.202,Z 826.7,A -85,B 0,C 180,E1 -18839.852,E2 -18839.852} C_VEL
LIN {X 0,Y 264.527,Z 818.113,A -85,B 0,C 180,E1 -18842.097,E2 -18842.097} C_VEL
LIN {X 0,Y 268.271,Z 808.324,A -85,B 0,C 180,E1 -18844.279,E2 -18844.279} C_VEL
LIN {X 0,Y 272.48,Z 797.099,A -85,B 0,C 180,E1 -18846.386,E2 -18846.386} C_VEL
LIN {X 0,Y 276.247,Z 786.399,A -85,B 0,C 180,E1 -18848.092,E2 -18848.092} C_VEL
LIN {X 0,Y 279.86,Z 775.429,A -85,B 0,C 180,E1 -18849.585,E2 -18849.585} C_VEL
LIN {X 0,Y 283.188,Z 764.298,A -85,B 0,C 180,E1 -18850.885,E2 -18850.885} C_VEL
LIN {X 0,Y 286.261,Z 753.144,A -85,B 0,C 180,E1 -18851.99,E2 -18851.99} C_VEL
LIN {X 0,Y 289.226,Z 741.016,A -85,B 0,C 180,E1 -18853.004,E2 -18853.004} C_VEL
LIN {X 0,Y 291.677,Z 729.576,A -85,B 0,C 180,E1 -18853.806,E2 -18853.806} C_VEL
LIN {X 0,Y 294.179,Z 715.953,A -85,B 0,C 180,E1 -18854.568,E2 -18854.568} C_VEL
LIN {X 0,Y 296.148,Z 702.586,A -85,B 0,C 180,E1 -18855.15,E2 -18855.15} C_VEL
LIN {X 0,Y 297.586,Z 689.133,A -85,B 0,C 180,E1 -18855.593,E2 -18855.593} C_VEL
LIN {X 0,Y 299.766,Z 653.639,A -85,B 0,C 180,E1 -18856.434,E2 -18856.434} C_VEL
LIN {X 0,Y 304.829,Z 564.515,A -85,B 0,C 180,E1 -18858.451,E2 -18858.451} C_VEL
LIN {X 0,Y 298.675,Z 550.938,A -85,B 0,C 180,E1 -18860.287,E2 -18860.287} C_VEL
LIN {X 0,Y 291.548,Z 536.606,A -85,B 0,C 180,E1 -18862.554,E2 -18862.554} C_VEL
LIN {X 0,Y 284.329,Z 523.759,A -85,B 0,C 180,E1 -18865.029,E2 -18865.029} C_VEL
LIN {X 0,Y 277.831,Z 513.205,A -85,B 0,C 180,E1 -18867.469,E2 -18867.469} C_VEL
LIN {X 0,Y 273.99,Z 507.38,A -85,B 0,C 180,E1 -18869.028,E2 -18869.028} C_VEL
LIN {X 0,Y 270.566,Z 502.922,A -85,B 0,C 180,E1 -18870.481,E2 -18870.481} C_VEL
LIN {X 0,Y 267.674,Z 499.051,A -85,B 0,C 180,E1 -18871.796,E2 -18871.796} C_VEL
LIN {X 0,Y 264.495,Z 495.482,A -85,B 0,C 180,E1 -18873.306,E2 -18873.306} C_VEL
LIN {X 0,Y 263.236,Z 493.534,A -85,B 0,C 180,E1 -18873.969,E2 -18873.969} C_VEL
LIN {X 0,Y 260.574,Z 491.071,A -85,B 0,C 180,E1 -18875.34,E2 -18875.34} C_VEL
LIN {X 0,Y 258.804,Z 488.266,A -85,B 0,C 180,E1 -18876.387,E2 -18876.387} C_VEL
LIN {X 0,Y 256.118,Z 486.165,A -85,B 0,C 180,E1 -18877.939,E2 -18877.939} C_VEL
LIN {X 0,Y 254.414,Z 483.32,A -85,B 0,C 180,E1 -18879.114,E2 -18879.114} C_VEL
LIN {X 0,Y 253.512,Z 482.358,A -85,B 0,C 180,E1 -18879.724,E2 -18879.724} C_VEL
LIN {X 0,Y 250.678,Z 480.258,A -85,B 0,C 180,E1 -18881.72,E2 -18881.72} C_VEL
LIN {X 0,Y 249.456,Z 477.896,A -85,B 0,C 180,E1 -18882.878,E2 -18882.878} C_VEL
LIN {X 0,Y 249.231,Z 476.736,A -85,B 0,C 180,E1 -18883.966,E2 -18883.966} C_VEL
LIN {X 0,Y 249.239,Z 476.681,A -85,B 0,C 180,E1 -18888.616,E2 -18888.616} C_VEL
LIN {X 0,Y 249.45,Z 476.638,A -85,B 0,C 180,E1 -18891.902,E2 -18891.902} C_VEL
LIN {X 0,Y 249.291,Z 476.664,A -85,B 0,C 180,E1 -18895.148,E2 -18895.148} C_VEL
LIN {X 0,Y 249.67,Z 476.627,A -85,B 0,C 180,E1 -18898.387,E2 -18898.387} C_VEL
LIN {X 0,Y 249.67,Z 476.606,A -85,B 0,C 180,E1 -18901.613,E2 -18901.613} C_VEL
LIN {X 0,Y 249.444,Z 476.634,A -85,B 0,C 180,E1 -18906.727,E2 -18906.727} C_VEL
LIN {X 0,Y 249.384,Z 476.651,A -85,B 0,C 180,E1 -18909.734,E2 -18909.734} C_VEL
LIN {X 0,Y 249.192,Z 476.676,A -85,B 0,C 180,E1 -18914.704,E2 -18914.704} C_VEL
LIN {X 0,Y 249.222,Z 476.977,A -85,B 0,C 180,E1 -18916.758,E2 -18916.758} C_VEL
LIN {X 0,Y 249.493,Z 478.091,A -85,B 0,C 180,E1 -18917.626,E2 -18917.626} C_VEL
LIN {X 0,Y 250.803,Z 480.466,A -85,B 0,C 180,E1 -18918.799,E2 -18918.799} C_VEL
LIN {X 0,Y 253.319,Z 482.315,A -85,B 0,C 180,E1 -18920.571,E2 -18920.571} C_VEL
LIN {X 0,Y 254.301,Z 483.136,A -85,B 0,C 180,E1 -18921.222,E2 -18921.222} C_VEL
LIN {X 0,Y 255.829,Z 485.905,A -85,B 0,C 180,E1 -18922.299,E2 -18922.299} C_VEL
LIN {X 0,Y 258.486,Z 488.074,A -85,B 0,C 180,E1 -18923.855,E2 -18923.855} C_VEL
LIN {X 0,Y 259.188,Z 488.742,A -85,B 0,C 180,E1 -18924.252,E2 -18924.252} C_VEL
LIN {X 0,Y 261.332,Z 491.92,A -85,B 0,C 180,E1 -18925.485,E2 -18925.485} C_VEL
LIN {X 0,Y 263.675,Z 494.132,A -85,B 0,C 180,E1 -18926.676,E2 -18926.676} C_VEL
LIN {X 0,Y 266.177,Z 497.605,A -85,B 0,C 180,E1 -18927.936,E2 -18927.936} C_VEL
LIN {X 0,Y 267.868,Z 499.393,A -85,B 0,C 180,E1 -18928.715,E2 -18928.715} C_VEL
LIN {X 0,Y 270.841,Z 503.204,A -85,B 0,C 180,E1 -18930.051,E2 -18930.051} C_VEL
LIN {X 0,Y 275.743,Z 509.556,A -85,B 0,C 180,E1 -18932.09,E2 -18932.09} C_VEL
LIN {X 0,Y 286.477,Z 523.303,A -85,B 0,C 180,E1 -18935.972,E2 -18935.972} C_VEL
LIN {X 0,Y 293.185,Z 530.297,A -85,B 0,C 180,E1 -18938.028,E2 -18938.028} C_VEL
LIN {X 0,Y 299.447,Z 536.358,A -85,B 0,C 180,E1 -18939.891,E2 -18939.891} C_VEL
LIN {X 0,Y 303.246,Z 539.763,A -85,B 0,C 180,E1 -18941.066,E2 -18941.066} C_VEL
LIN {X 0,Y 308.314,Z 544.304,A -85,B 0,C 180,E1 -18942.729,E2 -18942.729} C_VEL
LIN {X 0,Y 313.999,Z 549.704,A -85,B 0,C 180,E1 -18944.733,E2 -18944.733} C_VEL
LIN {X 0,Y 317.884,Z 553.443,A -85,B 0,C 180,E1 -18946.229,E2 -18946.229} C_VEL
LIN {X 0,Y 322.03,Z 557.246,A -85,B 0,C 180,E1 -18947.903,E2 -18947.903} C_VEL
LIN {X 0,Y 327.186,Z 562.436,A -85,B 0,C 180,E1 -18950.063,E2 -18950.063} C_VEL
LIN {X 0,Y 330.058,Z 564.972,A -85,B 0,C 180,E1 -18951.291,E2 -18951.291} C_VEL
LIN {X 0,Y 334.544,Z 569.341,A -85,B 0,C 180,E1 -18953.271,E2 -18953.271} C_VEL
LIN {X 0,Y 337.539,Z 571.937,A -85,B 0,C 180,E1 -18954.621,E2 -18954.621} C_VEL
LIN {X 0,Y 341.772,Z 575.987,A -85,B 0,C 180,E1 -18956.63,E2 -18956.63} C_VEL
LIN {X 0,Y 345.038,Z 578.619,A -85,B 0,C 180,E1 -18958.206,E2 -18958.206} C_VEL
LIN {X 0,Y 348.696,Z 582.156,A -85,B 0,C 180,E1 -18960.073,E2 -18960.073} C_VEL
LIN {X 0,Y 352.569,Z 585.288,A -85,B 0,C 180,E1 -18962.143,E2 -18962.143} C_VEL
LIN {X 0,Y 356.607,Z 589.319,A -85,B 0,C 180,E1 -18964.487,E2 -18964.487} C_VEL
LIN {X 0,Y 360.842,Z 592.395,A -85,B 0,C 180,E1 -18967.075,E2 -18967.075} C_VEL
LIN {X 0,Y 363.916,Z 595.546,A -85,B 0,C 180,E1 -18969.235,E2 -18969.235} C_VEL
LIN {X 0,Y 367.282,Z 598.008,A -85,B 0,C 180,E1 -18971.731,E2 -18971.731} C_VEL
LIN {X 0,Y 369.42,Z 599.313,A -85,B 0,C 180,E1 -18973.478,E2 -18973.478} C_VEL
LIN {X 0,Y 371.755,Z 602.027,A -85,B 0,C 180,E1 -18975.773,E2 -18975.773} C_VEL
LIN {X 0,Y 374.213,Z 604.128,A -85,B 0,C 180,E1 -18978.549,E2 -18978.549} C_VEL
LIN {X 0,Y 375.982,Z 605.025,A -85,B 0,C 180,E1 -18980.905,E2 -18980.905} C_VEL
LIN {X 0,Y 377.482,Z 605.766,A -85,B 0,C 180,E1 -18983.586,E2 -18983.586} C_VEL
LIN {X 0,Y 378.302,Z 606.332,A -85,B 0,C 180,E1 -18985.738,E2 -18985.738} C_VEL
LIN {X 0,Y 378.827,Z 606.512,A -85,B 0,C 180,E1 -18987.874,E2 -18987.874} C_VEL
LIN {X 0,Y 379.014,Z 606.578,A -85,B 0,C 180,E1 -18990,E2 -18990} C_VEL
LIN {X 0,Y 378.827,Z 606.512,A -85,B 0,C 180,E1 -18992.126,E2 -18992.126} C_VEL
LIN {X 0,Y 378.144,Z 606.223,A -85,B 0,C 180,E1 -18994.77,E2 -18994.77} C_VEL
LIN {X 0,Y 376.937,Z 605.518,A -85,B 0,C 180,E1 -18997.499,E2 -18997.499} C_VEL
LIN {X 0,Y 375.115,Z 604.653,A -85,B 0,C 180,E1 -19000.326,E2 -19000.326} C_VEL
LIN {X 0,Y 372.988,Z 603.154,A -85,B 0,C 180,E1 -19002.888,E2 -19002.888} C_VEL
LIN {X 0,Y 370.675,Z 600.867,A -85,B 0,C 180,E1 -19005.32,E2 -19005.32} C_VEL
LIN {X 0,Y 368.898,Z 598.829,A -85,B 0,C 180,E1 -19006.983,E2 -19006.983} C_VEL
LIN {X 0,Y 365.884,Z 597.077,A -85,B 0,C 180,E1 -19009.331,E2 -19009.331} C_VEL
LIN {X 0,Y 362.455,Z 594.175,A -85,B 0,C 180,E1 -19011.803,E2 -19011.803} C_VEL
LIN {X 0,Y 360.024,Z 591.656,A -85,B 0,C 180,E1 -19013.441,E2 -19013.441} C_VEL
LIN {X 0,Y 356.088,Z 588.846,A -85,B 0,C 180,E1 -19015.826,E2 -19015.826} C_VEL
LIN {X 0,Y 352.324,Z 585.053,A -85,B 0,C 180,E1 -19017.994,E2 -19017.994} C_VEL
LIN {X 0,Y 347.266,Z 580.946,A -85,B 0,C 180,E1 -19020.652,E2 -19020.652} C_VEL
LIN {X 0,Y 343.611,Z 577.364,A -85,B 0,C 180,E1 -19022.509,E2 -19022.509} C_VEL
LIN {X 0,Y 338.865,Z 573.351,A -85,B 0,C 180,E1 -19024.746,E2 -19024.746} C_VEL
LIN {X 0,Y 335.431,Z 570.016,A -85,B 0,C 180,E1 -19026.334,E2 -19026.334} C_VEL
LIN {X 0,Y 330.664,Z 565.664,A -85,B 0,C 180,E1 -19028.445,E2 -19028.445} C_VEL
LIN {X 0,Y 328.118,Z 563.167,A -85,B 0,C 180,E1 -19029.549,E2 -19029.549} C_VEL
LIN {X 0,Y 323.513,Z 558.844,A -85,B 0,C 180,E1 -19031.482,E2 -19031.482} C_VEL
LIN {X 0,Y 320.406,Z 555.854,A -85,B 0,C 180,E1 -19032.762,E2 -19032.762} C_VEL
LIN {X 0,Y 314.002,Z 549.684,A -85,B 0,C 180,E1 -19035.267,E2 -19035.267} C_VEL
LIN {X 0,Y 309.138,Z 544.985,A -85,B 0,C 180,E1 -19036.999,E2 -19036.999} C_VEL
LIN {X 0,Y 303.555,Z 540.089,A -85,B 0,C 180,E1 -19038.833,E2 -19038.833} C_VEL
LIN {X 0,Y 299.78,Z 536.618,A -85,B 0,C 180,E1 -19040.01,E2 -19040.01} C_VEL
LIN {X 0,Y 294.647,Z 531.661,A -85,B 0,C 180,E1 -19041.546,E2 -19041.546} C_VEL
LIN {X 0,Y 288.436,Z 525.467,A -85,B 0,C 180,E1 -19043.402,E2 -19043.402} C_VEL
LIN {X 0,Y 282.737,Z 518.75,A -85,B 0,C 180,E1 -19045.294,E2 -19045.294} C_VEL
LIN {X 0,Y 274.023,Z 507.32,A -85,B 0,C 180,E1 -19048.604,E2 -19048.604} C_VEL
LIN {X 0,Y 270.847,Z 503.205,A -85,B 0,C 180,E1 -19049.946,E2 -19049.946} C_VEL
LIN {X 0,Y 267.779,Z 499.249,A -85,B 0,C 180,E1 -19051.328,E2 -19051.328} C_VEL
LIN {X 0,Y 264.305,Z 495.22,A -85,B 0,C 180,E1 -19052.987,E2 -19052.987} C_VEL
LIN {X 0,Y 263.166,Z 493.448,A -85,B 0,C 180,E1 -19053.589,E2 -19053.589} C_VEL
LIN {X 0,Y 260.338,Z 490.707,A -85,B 0,C 180,E1 -19055.06,E2 -19055.06} C_VEL
LIN {X 0,Y 258.82,Z 488.252,A -85,B 0,C 180,E1 -19055.965,E2 -19055.965} C_VEL
LIN {X 0,Y 256.121,Z 486.26,A -85,B 0,C 180,E1 -19057.515,E2 -19057.515} C_VEL
LIN {X 0,Y 254.484,Z 483.598,A -85,B 0,C 180,E1 -19058.635,E2 -19058.635} C_VEL
LIN {X 0,Y 253.903,Z 482.656,A -85,B 0,C 180,E1 -19059.051,E2 -19059.051} C_VEL
LIN {X 0,Y 251.055,Z 480.714,A -85,B 0,C 180,E1 -19061.009,E2 -19061.009} C_VEL
LIN {X 0,Y 249.572,Z 478.393,A -85,B 0,C 180,E1 -19062.274,E2 -19062.274} C_VEL
LIN {X 0,Y 249.25,Z 477.159,A -85,B 0,C 180,E1 -19063.012,E2 -19063.012} C_VEL
LIN {X 0,Y 249.237,Z 476.741,A -85,B 0,C 180,E1 -19063.622,E2 -19063.622} C_VEL
LIN {X 0,Y 249.247,Z 476.66,A -85,B 0,C 180,E1 -19068.617,E2 -19068.617} C_VEL
LIN {X 0,Y 249.474,Z 476.646,A -85,B 0,C 180,E1 -19071.903,E2 -19071.903} C_VEL
LIN {X 0,Y 249.431,Z 476.654,A -85,B 0,C 180,E1 -19076.77,E2 -19076.77} C_VEL
LIN {X 0,Y 249.716,Z 476.613,A -85,B 0,C 180,E1 -19080,E2 -19080} C_VEL
LIN {X 0,Y 249.429,Z 476.64,A -85,B 0,C 180,E1 -19083.231,E2 -19083.231} C_VEL
LIN {X 0,Y 249.449,Z 476.656,A -85,B 0,C 180,E1 -19086.471,E2 -19086.471} C_VEL
LIN {X 0,Y 249.338,Z 476.656,A -85,B 0,C 180,E1 -19089.737,E2 -19089.737} C_VEL
LIN {X 0,Y 249.192,Z 476.677,A -85,B 0,C 180,E1 -19094.704,E2 -19094.704} C_VEL
LIN {X 0,Y 249.249,Z 476.99,A -85,B 0,C 180,E1 -19096.378,E2 -19096.378} C_VEL
LIN {X 0,Y 249.57,Z 478.239,A -85,B 0,C 180,E1 -19097.289,E2 -19097.289} C_VEL
LIN {X 0,Y 250.928,Z 480.512,A -85,B 0,C 180,E1 -19098.472,E2 -19098.472} C_VEL
LIN {X 0,Y 254.304,Z 483.085,A -85,B 0,C 180,E1 -19100.804,E2 -19100.804} C_VEL
LIN {X 0,Y 255.969,Z 486.021,A -85,B 0,C 180,E1 -19101.969,E2 -19101.969} C_VEL
LIN {X 0,Y 258.47,Z 488.094,A -85,B 0,C 180,E1 -19103.432,E2 -19103.432} C_VEL
LIN {X 0,Y 259.196,Z 488.742,A -85,B 0,C 180,E1 -19103.84,E2 -19103.84} C_VEL
LIN {X 0,Y 261.271,Z 491.906,A -85,B 0,C 180,E1 -19105.04,E2 -19105.04} C_VEL
LIN {X 0,Y 263.663,Z 494.079,A -85,B 0,C 180,E1 -19106.252,E2 -19106.252} C_VEL
LIN {X 0,Y 266.2,Z 497.615,A -85,B 0,C 180,E1 -19107.53,E2 -19107.53} C_VEL
LIN {X 0,Y 267.851,Z 499.354,A -85,B 0,C 180,E1 -19108.29,E2 -19108.29} C_VEL
LIN {X 0,Y 270.869,Z 503.236,A -85,B 0,C 180,E1 -19109.648,E2 -19109.648} C_VEL
LIN {X 0,Y 275.68,Z 509.882,A -85,B 0,C 180,E1 -19111.669,E2 -19111.669} C_VEL
LIN {X 0,Y 281.601,Z 519.213,A -85,B 0,C 180,E1 -19113.974,E2 -19113.974} C_VEL
LIN {X 0,Y 288.623,Z 531.251,A -85,B 0,C 180,E1 -19116.469,E2 -19116.469} C_VEL
LIN {X 0,Y 295.881,Z 545.192,A -85,B 0,C 180,E1 -19118.846,E2 -19118.846} C_VEL
LIN {X 0,Y 301.34,Z 556.549,A -85,B 0,C 180,E1 -19120.516,E2 -19120.516} C_VEL
LIN {X 0,Y 301.978,Z 559.409,A -85,B 0,C 180,E1 -19120.758,E2 -19120.758} C_VEL
LIN {X 0,Y 301.815,Z 563.938,A -85,B 0,C 180,E1 -19120.884,E2 -19120.884} C_VEL
LIN {X 0,Y 299.497,Z 576.291,A -85,B 0,C 180,E1 -19120.816,E2 -19120.816} C_VEL
LIN {X 0,Y 299.387,Z 577.69,A -85,B 0,C 180,E1 -19120.842,E2 -19120.842} C_VEL
LIN {X 0,Y 292.916,Z 686.199,A -85,B 0,C 180,E1 -19123.341,E2 -19123.341} C_VEL
LIN {X 0,Y 291.43,Z 700.377,A -85,B 0,C 180,E1 -19123.785,E2 -19123.785} C_VEL
LIN {X 0,Y 289.506,Z 713.444,A -85,B 0,C 180,E1 -19124.327,E2 -19124.327} C_VEL
LIN {X 0,Y 287.203,Z 726.163,A -85,B 0,C 180,E1 -19125.012,E2 -19125.012} C_VEL
LIN {X 0,Y 284.622,Z 738.525,A -85,B 0,C 180,E1 -19125.852,E2 -19125.852} C_VEL
LIN {X 0,Y 281.934,Z 749.451,A -85,B 0,C 180,E1 -19126.725,E2 -19126.725} C_VEL
LIN {X 0,Y 278.731,Z 761.088,A -85,B 0,C 180,E1 -19127.831,E2 -19127.831} C_VEL
LIN {X 0,Y 274.82,Z 773.914,A -85,B 0,C 180,E1 -19129.3,E2 -19129.3} C_VEL
LIN {X 0,Y 271.059,Z 785.044,A -85,B 0,C 180,E1 -19130.804,E2 -19130.804} C_VEL
LIN {X 0,Y 267.389,Z 795.35,A -85,B 0,C 180,E1 -19132.444,E2 -19132.444} C_VEL
LIN {X 0,Y 263.777,Z 804.561,A -85,B 0,C 180,E1 -19134.116,E2 -19134.116} C_VEL
LIN {X 0,Y 259.688,Z 814.767,A -85,B 0,C 180,E1 -19136.304,E2 -19136.304} C_VEL
LIN {X 0,Y 256.025,Z 823.726,A -85,B 0,C 180,E1 -19138.564,E2 -19138.564} C_VEL
LIN {X 0,Y 252.737,Z 831.618,A -85,B 0,C 180,E1 -19140.881,E2 -19140.881} C_VEL
LIN {X 0,Y 249.807,Z 838.582,A -85,B 0,C 180,E1 -19143.248,E2 -19143.248} C_VEL
LIN {X 0,Y 247.145,Z 845.117,A -85,B 0,C 180,E1 -19145.842,E2 -19145.842} C_VEL
LIN {X 0,Y 244.604,Z 851.677,A -85,B 0,C 180,E1 -19148.952,E2 -19148.952} C_VEL
